KUKA KRL program: MyProgram_003().src

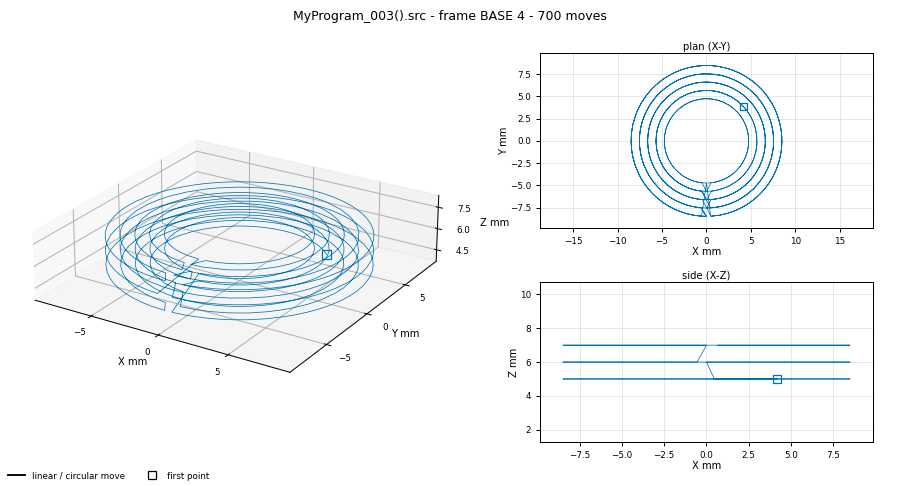
[picture p0: tool path of MyProgram_003().src in frame BASE 4, 700 of 700 moves have a stored position in this frame; points joined in program order, loops and branches not executed]
&ACCESS RVP
&REL 1
&PARAM TEMPLATE = C:\KRC\Roboter\Template\vorgabe
&PARAM EDITMASK = *
DEF MyProgram_003()
; ---- Setting reference (Base) ----
$BASE = BASE_DATA[4]

; --------------------------
; ---- Setting tool (TCP) ----
$TOOL = TOOL_DATA[3]
; --------------------------

$VEL.CP = VEL_APROX_PRINT
Startdeposition()
$VEL.CP = VEL_PRINT
LIN {X 4.1608,Y 3.8743,Z 5,A -2.5016,B 0,C 0,E1 0.1598,E2 90.072} C_DIS
LIN {X 3.5816,Y 4.4156,Z 5,A -2.5001,B 0,C 0,E1 0.1598,E2 90.072} C_DIS
LIN {X 2.9315,Y 4.8693,Z 5,A -2.5049,B 0,C 0,E1 0.1598,E2 90.0721} C_DIS
LIN {X 2.2263,Y 5.2312,Z 5,A -2.5157,B 0,C 0,E1 0.1598,E2 90.0721} C_DIS
LIN {X 1.4771,Y 5.4901,Z 5,A -2.5324,B 0,C 0,E1 0.1598,E2 90.0721} C_DIS
LIN {X 0.6988,Y 5.6397,Z 5,A -2.5548,B 0,C 0,E1 0.1598,E2 90.0721} C_DIS
LIN {X -0.0924,Y 5.6815,Z 5,A -2.5823,B 0,C 0,E1 0.1598,E2 90.0721} C_DIS
LIN {X -0.8823,Y 5.6159,Z 5,A -2.6142,B 0,C 0,E1 0.1598,E2 90.0721} C_DIS
LIN {X -1.6551,Y 5.4395,Z 5,A -2.6501,B 0,C 0,E1 0.1598,E2 90.0721} C_DIS
LIN {X -2.3959,Y 5.1568,Z 5,A -2.6893,B 0,C 0,E1 0.1598,E2 90.072} C_DIS
LIN {X -3.0893,Y 4.7724,Z 5,A -2.7311,B 0,C 0,E1 0.1598,E2 90.0719} C_DIS
LIN {X -3.8738,Y 4.1671,Z 5,A -2.7853,B 0,C 0,E1 0.1598,E2 90.0717} C_DIS
LIN {X -4.6268,Y 3.3119,Z 5,A -2.8489,B 0,C 0,E1 0.1598,E2 90.0714} C_DIS
LIN {X -5.1518,Y 2.4055,Z 5,A -2.9064,B 0,C 0,E1 0.1598,E2 90.0714} C_DIS
LIN {X -5.5303,Y 1.34,Z 5,A -2.965,B 0,C 0,E1 0.1598,E2 90.0711} C_DIS
LIN {X -5.6376,Y 0.726,Z 5,A -2.9951,B 0,C 0,E1 0.1598,E2 90.0713} C_DIS
LIN {X -5.6838,Y -0.1031,Z 5,A -3.0316,B 0,C 0,E1 0.1598,E2 90.0712} C_DIS
LIN {X -5.609,Y -0.9301,Z 5,A -3.0637,B 0,C 0,E1 0.1598,E2 90.0712} C_DIS
LIN {X -5.4131,Y -1.7371,Z 5,A -3.0905,B 0,C 0,E1 0.1598,E2 90.0712} C_DIS
LIN {X -5.1008,Y -2.5065,Z 5,A -3.1115,B 0,C 0,E1 0.1598,E2 90.0712} C_DIS
LIN {X -4.6803,Y -3.2223,Z 5,A -3.1262,B 0,C 0,E1 0.1598,E2 90.0712} C_DIS
LIN {X -4.1611,Y -3.8701,Z 5,A -3.1345,B 0,C 0,E1 0.1598,E2 90.0712} C_DIS
LIN {X -3.3929,Y -4.5678,Z 5,A -3.1357,B 0,C 0,E1 0.1598,E2 90.0711} C_DIS
LIN {X -2.2029,Y -5.2456,Z 5,A -3.1207,B 0,C 0,E1 0.1598,E2 90.0711} C_DIS
LIN {X -1.3096,Y -5.5324,Z 5,A -3.1002,B 0,C 0,E1 0.1598,E2 90.0714} C_DIS
LIN {X -0.5693,Y -5.6561,Z 5,A -3.0783,B 0,C 0,E1 0.1598,E2 90.0714} C_DIS
LIN {X -0.5693,Y -5.6561,Z 5,A -3.0783,B 0,C 0,E1 0.1598,E2 90.0714} C_DIS
Enddeposition()
LIN {X -0.0404,Y -6.6236,Z 5,A -3.0988,B 0,C 0,E1 0.1598,E2 90.0703} C_DIS
Startdeposition()
$VEL.CP = VEL_PRINT
LIN {X -0.9259,Y -6.553,Z 5,A -3.1294,B 0,C 0,E1 0.1598,E2 90.0713} C_DIS
LIN {X -1.6231,Y -6.4161,Z 5,A -3.1492,B 0,C 0,E1 0.1598,E2 90.0713} C_DIS
LIN {X -2.3026,Y -6.2076,Z 5,A -3.1654,B 0,C 0,E1 0.1598,E2 90.0713} C_DIS
LIN {X -2.9544,Y -5.9244,Z 5,A -3.1773,B 0,C 0,E1 0.1598,E2 90.0713} C_DIS
LIN {X -3.5722,Y -5.5732,Z 5,A -3.1851,B 0,C 0,E1 0.1598,E2 90.0713} C_DIS
LIN {X -4.1491,Y -5.1583,Z 5,A -3.1887,B 0,C 0,E1 0.1598,E2 90.0713} C_DIS
LIN {X -4.6779,Y -4.6835,Z 5,A -3.1881,B 0,C 0,E1 0.1598,E2 90.0713} C_DIS
LIN {X -5.1529,Y -4.1549,Z 5,A -3.1832,B 0,C 0,E1 0.1598,E2 90.0712} C_DIS
LIN {X -5.5689,Y -3.5788,Z 5,A -3.1742,B 0,C 0,E1 0.1598,E2 90.0712} C_DIS
LIN {X -5.9215,Y -2.9616,Z 5,A -3.1611,B 0,C 0,E1 0.1598,E2 90.0712} C_DIS
LIN {X -6.202,Y -2.3087,Z 5,A -3.1439,B 0,C 0,E1 0.1598,E2 90.0712} C_DIS
LIN {X -6.4151,Y -1.6307,Z 5,A -3.1231,B 0,C 0,E1 0.1598,E2 90.0712} C_DIS
LIN {X -6.5528,Y -0.9336,Z 5,A -3.0988,B 0,C 0,E1 0.1598,E2 90.0712} C_DIS
LIN {X -6.6173,Y -0.2258,Z 5,A -3.0714,B 0,C 0,E1 0.1598,E2 90.0712} C_DIS
LIN {X -6.6026,Y 0.4846,Z 5,A -3.041,B 0,C 0,E1 0.1598,E2 90.0712} C_DIS
LIN {X -6.5102,Y 1.1893,Z 5,A -3.0079,B 0,C 0,E1 0.1598,E2 90.0713} C_DIS
LIN {X -6.3462,Y 1.8807,Z 5,A -2.9728,B 0,C 0,E1 0.1598,E2 90.0713} C_DIS
LIN {X -6.1101,Y 2.5511,Z 5,A -2.9359,B 0,C 0,E1 0.1598,E2 90.0714} C_DIS
LIN {X -5.8024,Y 3.1918,Z 5,A -2.8976,B 0,C 0,E1 0.1598,E2 90.0715} C_DIS
LIN {X -5.4264,Y 3.795,Z 5,A -2.8584,B 0,C 0,E1 0.1598,E2 90.0715} C_DIS
LIN {X -4.9862,Y 4.3528,Z 5,A -2.8187,B 0,C 0,E1 0.1598,E2 90.0717} C_DIS
LIN {X -4.4919,Y 4.8634,Z 5,A -2.779,B 0,C 0,E1 0.1598,E2 90.0717} C_DIS
LIN {X -3.9448,Y 5.317,Z 5,A -2.7398,B 0,C 0,E1 0.1598,E2 90.0718} C_DIS
LIN {X -3.3521,Y 5.7091,Z 5,A -2.7015,B 0,C 0,E1 0.1598,E2 90.0718} C_DIS
LIN {X -2.7203,Y 6.034,Z 5,A -2.6645,B 0,C 0,E1 0.1598,E2 90.072} C_DIS
LIN {X -2.0578,Y 6.2916,Z 5,A -2.6292,B 0,C 0,E1 0.1598,E2 90.072} C_DIS
LIN {X -1.372,Y 6.4783,Z 5,A -2.596,B 0,C 0,E1 0.1598,E2 90.072} C_DIS
LIN {X -0.6697,Y 6.587,Z 5,A -2.5656,B 0,C 0,E1 0.1598,E2 90.0721} C_DIS
LIN {X 0.0402,Y 6.6208,Z 5,A -2.5379,B 0,C 0,E1 0.1598,E2 90.0721} C_DIS
LIN {X 0.7496,Y 6.5788,Z 5,A -2.5135,B 0,C 0,E1 0.1598,E2 90.0722} C_DIS
LIN {X 1.4503,Y 6.4593,Z 5,A -2.4927,B 0,C 0,E1 0.1598,E2 90.0722} C_DIS
LIN {X 2.1342,Y 6.2657,Z 5,A -2.4756,B 0,C 0,E1 0.1598,E2 90.0722} C_DIS
LIN {X 2.7941,Y 6.0022,Z 5,A -2.4624,B 0,C 0,E1 0.1598,E2 90.0722} C_DIS
LIN {X 3.4211,Y 5.6677,Z 5,A -2.4534,B 0,C 0,E1 0.1598,E2 90.0722} C_DIS
LIN {X 4.0075,Y 5.2662,Z 5,A -2.4487,B 0,C 0,E1 0.1598,E2 90.0722} C_DIS
LIN {X 4.5492,Y 4.8063,Z 5,A -2.4481,B 0,C 0,E1 0.1598,E2 90.0722} C_DIS
LIN {X 5.0416,Y 4.2938,Z 5,A -2.4516,B 0,C 0,E1 0.1598,E2 90.0722} C_DIS
LIN {X 5.4696,Y 3.7264,Z 5,A -2.4598,B 0,C 0,E1 0.1598,E2 90.0722} C_DIS
LIN {X 5.8381,Y 3.1188,Z 5,A -2.4719,B 0,C 0,E1 0.1598,E2 90.0721} C_DIS
LIN {X 6.1397,Y 2.4754,Z 5,A -2.4881,B 0,C 0,E1 0.1598,E2 90.0721} C_DIS
LIN {X 6.3699,Y 1.8031,Z 5,A -2.508,B 0,C 0,E1 0.1598,E2 90.072} C_DIS
LIN {X 6.5278,Y 1.1101,Z 5,A -2.5316,B 0,C 0,E1 0.1598,E2 90.072} C_DIS
LIN {X 6.6079,Y 0.4039,Z 5,A -2.5586,B 0,C 0,E1 0.1598,E2 90.0719} C_DIS
LIN {X 6.6124,Y -0.3068,Z 5,A -2.5885,B 0,C 0,E1 0.1598,E2 90.0719} C_DIS
LIN {X 6.542,Y -1.0138,Z 5,A -2.6211,B 0,C 0,E1 0.1598,E2 90.0719} C_DIS
LIN {X 6.3948,Y -1.7092,Z 5,A -2.656,B 0,C 0,E1 0.1598,E2 90.0718} C_DIS
LIN {X 6.1754,Y -2.3851,Z 5,A -2.6928,B 0,C 0,E1 0.1598,E2 90.0718} C_DIS
LIN {X 5.884,Y -3.0334,Z 5,A -2.731,B 0,C 0,E1 0.1598,E2 90.0718} C_DIS
LIN {X 5.5246,Y -3.6466,Z 5,A -2.7702,B 0,C 0,E1 0.1598,E2 90.0717} C_DIS
LIN {X 5.1021,Y -4.2181,Z 5,A -2.81,B 0,C 0,E1 0.1598,E2 90.0717} C_DIS
LIN {X 4.6202,Y -4.7402,Z 5,A -2.8499,B 0,C 0,E1 0.1598,E2 90.0717} C_DIS
LIN {X 4.0856,Y -5.2087,Z 5,A -2.8894,B 0,C 0,E1 0.1598,E2 90.0717} C_DIS
LIN {X 3.5047,Y -5.6183,Z 5,A -2.9281,B 0,C 0,E1 0.1598,E2 90.0716} C_DIS
LIN {X 2.8824,Y -5.9615,Z 5,A -2.9655,B 0,C 0,E1 0.1598,E2 90.0716} C_DIS
LIN {X 2.2263,Y -6.2348,Z 5,A -3.0012,B 0,C 0,E1 0.1598,E2 90.0716} C_DIS
LIN {X 1.5451,Y -6.4376,Z 5,A -3.0348,B 0,C 0,E1 0.1598,E2 90.0716} C_DIS
LIN {X 0.846,Y -6.5644,Z 5,A -3.0658,B 0,C 0,E1 0.1598,E2 90.0715} C_DIS
LIN {X -0.0404,Y -6.6236,Z 5,A -3.1008,B 0,C 0,E1 0.1598,E2 90.0715} C_DIS
Enddeposition()
LIN {X -0.0404,Y -6.6236,Z 5,A -3.1008,B 0,C 0,E1 0.1598,E2 90.0715} C_DIS
Startdeposition()
$VEL.CP = VEL_PRINT
LIN {X 0.4586,Y -7.5414,Z 5,A -3.121,B 0,C 0,E1 0.1598,E2 90.0709} C_DIS
LIN {X 1.4877,Y -7.4091,Z 5,A -3.0782,B 0,C 0,E1 0.1598,E2 90.0714} C_DIS
LIN {X 2.3467,Y -7.1836,Z 5,A -3.0371,B 0,C 0,E1 0.1598,E2 90.0715} C_DIS
LIN {X 3.457,Y -6.7151,Z 5,A -2.9765,B 0,C 0,E1 0.1598,E2 90.0715} C_DIS
LIN {X 4.4391,Y -6.1176,Z 5,A -2.915,B 0,C 0,E1 0.1598,E2 90.0715} C_DIS
LIN {X 5.3005,Y -5.3806,Z 5,A -2.852,B 0,C 0,E1 0.1598,E2 90.0715} C_DIS
LIN {X 5.8569,Y -4.7686,Z 5,A -2.8057,B 0,C 0,E1 0.1598,E2 90.0716} C_DIS
LIN {X 6.3438,Y -4.0999,Z 5,A -2.7594,B 0,C 0,E1 0.1598,E2 90.0716} C_DIS
LIN {X 6.8478,Y -3.1971,Z 5,A -2.7023,B 0,C 0,E1 0.1598,E2 90.0715} C_DIS
LIN {X 7.2249,Y -2.2147,Z 5,A -2.6467,B 0,C 0,E1 0.1598,E2 90.0715} C_DIS
LIN {X 7.5046,Y -0.888,Z 5,A -2.5797,B 0,C 0,E1 0.1598,E2 90.0712} C_DIS
LIN {X 7.5564,Y 0.1077,Z 5,A -2.536,B 0,C 0,E1 0.1598,E2 90.0717} C_DIS
LIN {X 7.4656,Y 1.1496,Z 5,A -2.495,B 0,C 0,E1 0.1598,E2 90.0717} C_DIS
LIN {X 7.2089,Y 2.2659,Z 5,A -2.4571,B 0,C 0,E1 0.1598,E2 90.0716} C_DIS
LIN {X 6.8696,Y 3.1485,Z 5,A -2.4324,B 0,C 0,E1 0.1598,E2 90.0719} C_DIS
LIN {X 6.2798,Y 4.2042,Z 5,A -2.4093,B 0,C 0,E1 0.1598,E2 90.0718} C_DIS
LIN {X 5.6133,Y 5.0619,Z 5,A -2.3977,B 0,C 0,E1 0.1598,E2 90.0719} C_DIS
LIN {X 4.7836,Y 5.8452,Z 5,A -2.3952,B 0,C 0,E1 0.1598,E2 90.0719} C_DIS
LIN {X 3.9189,Y 6.4611,Z 5,A -2.4012,B 0,C 0,E1 0.1598,E2 90.0721} C_DIS
LIN {X 2.5264,Y 7.1223,Z 5,A -2.4246,B 0,C 0,E1 0.1598,E2 90.0721} C_DIS
LIN {X 1.6107,Y 7.3833,Z 5,A -2.4476,B 0,C 0,E1 0.1598,E2 90.0723} C_DIS
LIN {X -0.1184,Y 7.5562,Z 5,A -2.5042,B 0,C 0,E1 0.1598,E2 90.0723} C_DIS
LIN {X -1.2622,Y 7.4509,Z 5,A -2.5509,B 0,C 0,E1 0.1598,E2 90.0722} C_DIS
LIN {X -2.8172,Y 7.0134,Z 5,A -2.6267,B 0,C 0,E1 0.1598,E2 90.072} C_DIS
LIN {X -3.9999,Y 6.411,Z 5,A -2.6956,B 0,C 0,E1 0.1598,E2 90.0718} C_DIS
LIN {X -4.7613,Y 5.8698,Z 5,A -2.7464,B 0,C 0,E1 0.1598,E2 90.0718} C_DIS
LIN {X -5.6287,Y 5.0444,Z 5,A -2.813,B 0,C 0,E1 0.1598,E2 90.0715} C_DIS
LIN {X -6.3509,Y 4.0973,Z 5,A -2.8793,B 0,C 0,E1 0.1598,E2 90.0713} C_DIS
LIN {X -6.9039,Y 3.0748,Z 5,A -2.9426,B 0,C 0,E1 0.1598,E2 90.0711} C_DIS
LIN {X -7.2823,Y 2.0215,Z 5,A -3.0008,B 0,C 0,E1 0.1598,E2 90.0711} C_DIS
LIN {X -7.4591,Y 1.1875,Z 5,A -3.0426,B 0,C 0,E1 0.1598,E2 90.0711} C_DIS
LIN {X -7.5506,Y 0.3399,Z 5,A -3.0815,B 0,C 0,E1 0.1598,E2 90.0711} C_DIS
LIN {X -7.5339,Y -0.5955,Z 5,A -3.1202,B 0,C 0,E1 0.1598,E2 90.071} C_DIS
LIN {X -7.3478,Y -1.7493,Z 5,A -3.1617,B 0,C 0,E1 0.1598,E2 90.0707} C_DIS
LIN {X -7.0494,Y -2.7246,Z 5,A -3.1919,B 0,C 0,E1 0.1598,E2 90.0707} C_DIS
LIN {X -6.5677,Y -3.731,Z 5,A -3.2166,B 0,C 0,E1 0.1598,E2 90.0707} C_DIS
LIN {X -5.9244,Y -4.6917,Z 5,A -3.2335,B 0,C 0,E1 0.1598,E2 90.0708} C_DIS
LIN {X -5.1075,Y -5.5639,Z 5,A -3.2403,B 0,C 0,E1 0.1598,E2 90.0708} C_DIS
LIN {X -4.2014,Y -6.2818,Z 5,A -3.2375,B 0,C 0,E1 0.1598,E2 90.071} C_DIS
LIN {X -3.3847,Y -6.7567,Z 5,A -3.2278,B 0,C 0,E1 0.1598,E2 90.0712} C_DIS
LIN {X -2.4228,Y -7.1598,Z 5,A -3.2096,B 0,C 0,E1 0.1598,E2 90.0712} C_DIS
LIN {X -1.5721,Y -7.3914,Z 5,A -3.1882,B 0,C 0,E1 0.1598,E2 90.0712} C_DIS
LIN {X -0.6387,Y -7.531,Z 5,A -3.1599,B 0,C 0,E1 0.1598,E2 90.0713} C_DIS
LIN {X -0.6387,Y -7.531,Z 5,A -3.1599,B 0,C 0,E1 0.1598,E2 90.0713} C_DIS
Enddeposition()
LIN {X -0.0485,Y -8.4894,Z 5,A -3.1779,B 0,C 0,E1 0.1598,E2 90.0702} C_DIS
Startdeposition()
$VEL.CP = VEL_PRINT
LIN {X -1.0658,Y -8.4207,Z 5,A -3.2134,B 0,C 0,E1 0.1598,E2 90.0712} C_DIS
LIN {X -1.8694,Y -8.2794,Z 5,A -3.2369,B 0,C 0,E1 0.1598,E2 90.0712} C_DIS
LIN {X -2.6556,Y -8.0613,Z 5,A -3.2565,B 0,C 0,E1 0.1598,E2 90.0712} C_DIS
LIN {X -3.4177,Y -7.7697,Z 5,A -3.2721,B 0,C 0,E1 0.1598,E2 90.0712} C_DIS
LIN {X -4.1482,Y -7.4061,Z 5,A -3.2835,B 0,C 0,E1 0.1598,E2 90.0712} C_DIS
LIN {X -4.8402,Y -6.9737,Z 5,A -3.2906,B 0,C 0,E1 0.1598,E2 90.0711} C_DIS
LIN {X -5.4872,Y -6.4765,Z 5,A -3.2933,B 0,C 0,E1 0.1598,E2 90.0711} C_DIS
LIN {X -6.2257,Y -5.7733,Z 5,A -3.2906,B 0,C 0,E1 0.1598,E2 90.0709} C_DIS
LIN {X -6.9713,Y -4.8425,Z 5,A -3.2785,B 0,C 0,E1 0.1598,E2 90.0707} C_DIS
LIN {X -7.3978,Y -4.1602,Z 5,A -3.2657,B 0,C 0,E1 0.1598,E2 90.071} C_DIS
LIN {X -7.7587,Y -3.441,Z 5,A -3.2486,B 0,C 0,E1 0.1598,E2 90.071} C_DIS
LIN {X -8.0498,Y -2.691,Z 5,A -3.2277,B 0,C 0,E1 0.1598,E2 90.071} C_DIS
LIN {X -8.268,Y -1.9165,Z 5,A -3.2031,B 0,C 0,E1 0.1598,E2 90.071} C_DIS
LIN {X -8.4122,Y -1.125,Z 5,A -3.1751,B 0,C 0,E1 0.1598,E2 90.071} C_DIS
LIN {X -8.4813,Y -0.3234,Z 5,A -3.144,B 0,C 0,E1 0.1598,E2 90.071} C_DIS
LIN {X -8.4491,Y 0.8445,Z 5,A -3.0933,B 0,C 0,E1 0.1598,E2 90.0708} C_DIS
LIN {X -8.2788,Y 1.8895,Z 5,A -3.0432,B 0,C 0,E1 0.1598,E2 90.071} C_DIS
LIN {X -7.9502,Y 2.9764,Z 5,A -2.9854,B 0,C 0,E1 0.1598,E2 90.071} C_DIS
LIN {X -7.621,Y 3.7394,Z 5,A -2.9415,B 0,C 0,E1 0.1598,E2 90.0713} C_DIS
LIN {X -7.2187,Y 4.4667,Z 5,A -2.8961,B 0,C 0,E1 0.1598,E2 90.0714} C_DIS
LIN {X -6.7474,Y 5.151,Z 5,A -2.85,B 0,C 0,E1 0.1598,E2 90.0715} C_DIS
LIN {X -6.2111,Y 5.7858,Z 5,A -2.8036,B 0,C 0,E1 0.1598,E2 90.0716} C_DIS
LIN {X -5.615,Y 6.3648,Z 5,A -2.7573,B 0,C 0,E1 0.1598,E2 90.0717} C_DIS
LIN {X -4.9653,Y 6.8829,Z 5,A -2.7116,B 0,C 0,E1 0.1598,E2 90.0718} C_DIS
LIN {X -4.2682,Y 7.3351,Z 5,A -2.6668,B 0,C 0,E1 0.1598,E2 90.0719} C_DIS
LIN {X -3.5302,Y 7.7169,Z 5,A -2.6235,B 0,C 0,E1 0.1598,E2 90.072} C_DIS
LIN {X -2.7586,Y 8.0253,Z 5,A -2.5821,B 0,C 0,E1 0.1598,E2 90.072} C_DIS
LIN {X -1.9606,Y 8.2567,Z 5,A -2.5429,B 0,C 0,E1 0.1598,E2 90.0722} C_DIS
LIN {X -1.1438,Y 8.4093,Z 5,A -2.5063,B 0,C 0,E1 0.1598,E2 90.0722} C_DIS
LIN {X -0.3161,Y 8.4816,Z 5,A -2.4727,B 0,C 0,E1 0.1598,E2 90.0722} C_DIS
LIN {X 0.5148,Y 8.4729,Z 5,A -2.4424,B 0,C 0,E1 0.1598,E2 90.0723} C_DIS
LIN {X 1.3407,Y 8.3814,Z 5,A -2.4157,B 0,C 0,E1 0.1598,E2 90.0723} C_DIS
LIN {X 2.1537,Y 8.2095,Z 5,A -2.3929,B 0,C 0,E1 0.1598,E2 90.0723} C_DIS
LIN {X 2.9463,Y 7.9598,Z 5,A -2.3742,B 0,C 0,E1 0.1598,E2 90.0723} C_DIS
LIN {X 3.7106,Y 7.6339,Z 5,A -2.3597,B 0,C 0,E1 0.1598,E2 90.0723} C_DIS
LIN {X 4.4394,Y 7.2347,Z 5,A -2.3496,B 0,C 0,E1 0.1598,E2 90.0723} C_DIS
LIN {X 5.3674,Y 6.5808,Z 5,A -2.3429,B 0,C 0,E1 0.1598,E2 90.0722} C_DIS
LIN {X 6.1123,Y 5.8907,Z 5,A -2.3446,B 0,C 0,E1 0.1598,E2 90.0722} C_DIS
LIN {X 6.6465,Y 5.2788,Z 5,A -2.3508,B 0,C 0,E1 0.1598,E2 90.0722} C_DIS
LIN {X 7.1199,Y 4.6188,Z 5,A -2.3613,B 0,C 0,E1 0.1598,E2 90.0722} C_DIS
LIN {X 7.5283,Y 3.9167,Z 5,A -2.376,B 0,C 0,E1 0.1598,E2 90.0722} C_DIS
LIN {X 7.868,Y 3.1789,Z 5,A -2.3947,B 0,C 0,E1 0.1598,E2 90.0721} C_DIS
LIN {X 8.1958,Y 2.2181,Z 5,A -2.4231,B 0,C 0,E1 0.1598,E2 90.0717} C_DIS
LIN {X 8.4199,Y 1.0739,Z 5,A -2.4632,B 0,C 0,E1 0.1598,E2 90.0715} C_DIS
LIN {X 8.4832,Y 0.2891,Z 5,A -2.4946,B 0,C 0,E1 0.1598,E2 90.0719} C_DIS
LIN {X 8.4734,Y -0.4982,Z 5,A -2.5284,B 0,C 0,E1 0.1598,E2 90.0719} C_DIS
LIN {X 8.3355,Y -1.6188,Z 5,A -2.5807,B 0,C 0,E1 0.1598,E2 90.0715} C_DIS
LIN {X 8.077,Y -2.6093,Z 5,A -2.6324,B 0,C 0,E1 0.1598,E2 90.0715} C_DIS
LIN {X 7.7877,Y -3.3754,Z 5,A -2.6757,B 0,C 0,E1 0.1598,E2 90.0717} C_DIS
LIN {X 7.4261,Y -4.1102,Z 5,A -2.7202,B 0,C 0,E1 0.1598,E2 90.0717} C_DIS
LIN {X 6.9956,Y -4.8068,Z 5,A -2.7657,B 0,C 0,E1 0.1598,E2 90.0717} C_DIS
LIN {X 6.5,Y -5.4586,Z 5,A -2.8116,B 0,C 0,E1 0.1598,E2 90.0717} C_DIS
LIN {X 5.7223,Y -6.2741,Z 5,A -2.8746,B 0,C 0,E1 0.1598,E2 90.0714} C_DIS
LIN {X 4.878,Y -6.9455,Z 5,A -2.9342,B 0,C 0,E1 0.1598,E2 90.0714} C_DIS
LIN {X 4.1473,Y -7.4046,Z 5,A -2.9806,B 0,C 0,E1 0.1598,E2 90.0715} C_DIS
LIN {X 3.3736,Y -7.7869,Z 5,A -3.0252,B 0,C 0,E1 0.1598,E2 90.0715} C_DIS
LIN {X 2.5655,Y -8.0896,Z 5,A -3.0677,B 0,C 0,E1 0.1598,E2 90.0715} C_DIS
LIN {X 1.52,Y -8.3549,Z 5,A -3.1172,B 0,C 0,E1 0.1598,E2 90.0714} C_DIS
LIN {X 0.4661,Y -8.4736,Z 5,A -3.1609,B 0,C 0,E1 0.1598,E2 90.0714} C_DIS
LIN {X 0.4661,Y -8.4736,Z 5,A -3.1609,B 0,C 0,E1 0.1598,E2 90.0714} C_DIS
Enddeposition()
LIN {X 0.0002,Y -4.7527,Z 6,A -3.0051,B 0,C 0,E1 0.1598,E2 90.0603} C_DIS
Startdeposition()
$VEL.CP = VEL_PRINT
LIN {X 0.0002,Y -4.7527,Z 6,A -3.0108,B 0,C 0,E1 0.1598,E2 90.066} C_DIS
LIN {X 0.8436,Y -4.6754,Z 6,A -2.9814,B 0,C 0,E1 0.1598,E2 90.0709} C_DIS
LIN {X 1.5802,Y -4.479,Z 6,A -2.9466,B 0,C 0,E1 0.1598,E2 90.0716} C_DIS
LIN {X 2.1262,Y -4.2473,Z 6,A -2.9168,B 0,C 0,E1 0.1598,E2 90.0716} C_DIS
LIN {X 2.7108,Y -3.904,Z 6,A -2.8807,B 0,C 0,E1 0.1598,E2 90.0716} C_DIS
LIN {X 3.2384,Y -3.4779,Z 6,A -2.8433,B 0,C 0,E1 0.1598,E2 90.0716} C_DIS
LIN {X 3.7,Y -2.9815,Z 6,A -2.8052,B 0,C 0,E1 0.1598,E2 90.0717} C_DIS
LIN {X 4.0865,Y -2.4244,Z 6,A -2.7674,B 0,C 0,E1 0.1598,E2 90.0717} C_DIS
LIN {X 4.3892,Y -1.818,Z 6,A -2.7305,B 0,C 0,E1 0.1598,E2 90.0717} C_DIS
LIN {X 4.603,Y -1.1746,Z 6,A -2.6954,B 0,C 0,E1 0.1598,E2 90.0717} C_DIS
LIN {X 4.7242,Y -0.5078,Z 6,A -2.6627,B 0,C 0,E1 0.1598,E2 90.0717} C_DIS
LIN {X 4.7491,Y 0.1698,Z 6,A -2.633,B 0,C 0,E1 0.1598,E2 90.0718} C_DIS
LIN {X 4.6586,Y 0.9268,Z 6,A -2.6042,B 0,C 0,E1 0.1598,E2 90.0718} C_DIS
LIN {X 4.5069,Y 1.5002,Z 6,A -2.5856,B 0,C 0,E1 0.1598,E2 90.0719} C_DIS
LIN {X 4.2491,Y 2.1272,Z 6,A -2.5686,B 0,C 0,E1 0.1598,E2 90.0719} C_DIS
LIN {X 3.9029,Y 2.7102,Z 6,A -2.5567,B 0,C 0,E1 0.1598,E2 90.0719} C_DIS
LIN {X 3.4777,Y 3.2383,Z 6,A -2.55,B 0,C 0,E1 0.1598,E2 90.072} C_DIS
LIN {X 2.9815,Y 3.7002,Z 6,A -2.5488,B 0,C 0,E1 0.1598,E2 90.072} C_DIS
LIN {X 2.4242,Y 4.0861,Z 6,A -2.5531,B 0,C 0,E1 0.1598,E2 90.072} C_DIS
LIN {X 1.8178,Y 4.3889,Z 6,A -2.5627,B 0,C 0,E1 0.1598,E2 90.072} C_DIS
LIN {X 1.1746,Y 4.6027,Z 6,A -2.5774,B 0,C 0,E1 0.1598,E2 90.0721} C_DIS
LIN {X 0.5077,Y 4.7248,Z 6,A -2.5968,B 0,C 0,E1 0.1598,E2 90.0721} C_DIS
LIN {X -0.2544,Y 4.7428,Z 6,A -2.6242,B 0,C 0,E1 0.1598,E2 90.0721} C_DIS
LIN {X -0.8439,Y 4.6769,Z 6,A -2.6487,B 0,C 0,E1 0.1598,E2 90.0721} C_DIS
LIN {X -1.5001,Y 4.5068,Z 6,A -2.6801,B 0,C 0,E1 0.1598,E2 90.072} C_DIS
LIN {X -2.1271,Y 4.249,Z 6,A -2.714,B 0,C 0,E1 0.1598,E2 90.072} C_DIS
LIN {X -2.7104,Y 3.9033,Z 6,A -2.7501,B 0,C 0,E1 0.1598,E2 90.0719} C_DIS
LIN {X -3.2385,Y 3.4781,Z 6,A -2.7874,B 0,C 0,E1 0.1598,E2 90.0718} C_DIS
LIN {X -3.6997,Y 2.9813,Z 6,A -2.8253,B 0,C 0,E1 0.1598,E2 90.0717} C_DIS
LIN {X -4.0859,Y 2.4241,Z 6,A -2.863,B 0,C 0,E1 0.1598,E2 90.0717} C_DIS
LIN {X -4.3885,Y 1.8175,Z 6,A -2.8996,B 0,C 0,E1 0.1598,E2 90.0715} C_DIS
LIN {X -4.6022,Y 1.1744,Z 6,A -2.9346,B 0,C 0,E1 0.1598,E2 90.0715} C_DIS
LIN {X -4.7237,Y 0.5076,Z 6,A -2.9671,B 0,C 0,E1 0.1598,E2 90.0714} C_DIS
LIN {X -4.749,Y -0.1698,Z 6,A -2.9966,B 0,C 0,E1 0.1598,E2 90.0714} C_DIS
LIN {X -4.6753,Y -0.8437,Z 6,A -3.0223,B 0,C 0,E1 0.1598,E2 90.0714} C_DIS
LIN {X -4.5073,Y -1.5004,Z 6,A -3.0438,B 0,C 0,E1 0.1598,E2 90.0713} C_DIS
LIN {X -4.2474,Y -2.1265,Z 6,A -3.0606,B 0,C 0,E1 0.1598,E2 90.0713} C_DIS
LIN {X -3.9034,Y -2.7105,Z 6,A -3.0727,B 0,C 0,E1 0.1598,E2 90.0713} C_DIS
LIN {X -3.4778,Y -3.2384,Z 6,A -3.0793,B 0,C 0,E1 0.1598,E2 90.0713} C_DIS
LIN {X -2.9815,Y -3.7,Z 6,A -3.0806,B 0,C 0,E1 0.1598,E2 90.0713} C_DIS
LIN {X -2.4244,Y -4.0865,Z 6,A -3.0765,B 0,C 0,E1 0.1598,E2 90.0713} C_DIS
LIN {X -1.8178,Y -4.3887,Z 6,A -3.067,B 0,C 0,E1 0.1598,E2 90.0714} C_DIS
LIN {X -1.1745,Y -4.6023,Z 6,A -3.0524,B 0,C 0,E1 0.1598,E2 90.0714} C_DIS
LIN {X -0.5077,Y -4.725,Z 6,A -3.0332,B 0,C 0,E1 0.1598,E2 90.0715} C_DIS
LIN {X -0.5077,Y -4.725,Z 6,A -3.0332,B 0,C 0,E1 0.1598,E2 90.0715} C_DIS
Enddeposition()
LIN {X 0.0016,Y -5.6864,Z 6,A -3.0541,B 0,C 0,E1 0.1598,E2 90.0703} C_DIS
Startdeposition()
$VEL.CP = VEL_PRINT
LIN {X -0.9286,Y -5.6133,Z 6,A -3.0863,B 0,C 0,E1 0.1598,E2 90.0714} C_DIS
LIN {X -2.0374,Y -5.3126,Z 6,A -3.1142,B 0,C 0,E1 0.1598,E2 90.0714} C_DIS
LIN {X -3.1502,Y -4.7386,Z 6,A -3.1307,B 0,C 0,E1 0.1598,E2 90.0712} C_DIS
LIN {X -3.9721,Y -4.0673,Z 6,A -3.1325,B 0,C 0,E1 0.1598,E2 90.0712} C_DIS
LIN {X -4.5331,Y -3.43,Z 6,A -3.1262,B 0,C 0,E1 0.1598,E2 90.0712} C_DIS
LIN {X -4.9939,Y -2.717,Z 6,A -3.1131,B 0,C 0,E1 0.1598,E2 90.0712} C_DIS
LIN {X -5.3425,Y -1.9429,Z 6,A -3.0932,B 0,C 0,E1 0.1598,E2 90.0712} C_DIS
LIN {X -5.5724,Y -1.1256,Z 6,A -3.0672,B 0,C 0,E1 0.1598,E2 90.0712} C_DIS
LIN {X -5.6786,Y -0.2832,Z 6,A -3.0356,B 0,C 0,E1 0.1598,E2 90.0712} C_DIS
LIN {X -5.6579,Y 0.5657,Z 6,A -2.999,B 0,C 0,E1 0.1598,E2 90.0712} C_DIS
LIN {X -5.51,Y 1.4018,Z 6,A -2.9584,B 0,C 0,E1 0.1598,E2 90.0712} C_DIS
LIN {X -5.2388,Y 2.2064,Z 6,A -2.9146,B 0,C 0,E1 0.1598,E2 90.0714} C_DIS
LIN {X -4.852,Y 2.962,Z 6,A -2.8685,B 0,C 0,E1 0.1598,E2 90.0714} C_DIS
LIN {X -4.2219,Y 3.816,Z 6,A -2.8092,B 0,C 0,E1 0.1598,E2 90.0714} C_DIS
LIN {X -3.4205,Y 4.539,Z 6,A -2.7494,B 0,C 0,E1 0.1598,E2 90.0716} C_DIS
LIN {X -2.7779,Y 4.9589,Z 6,A -2.7082,B 0,C 0,E1 0.1598,E2 90.0719} C_DIS
LIN {X -2.0841,Y 5.2875,Z 6,A -2.6688,B 0,C 0,E1 0.1598,E2 90.0719} C_DIS
LIN {X -1.3526,Y 5.52,Z 6,A -2.632,B 0,C 0,E1 0.1598,E2 90.072} C_DIS
LIN {X -0.1317,Y 5.6882,Z 6,A -2.5799,B 0,C 0,E1 0.1598,E2 90.0721} C_DIS
LIN {X 0.8981,Y 5.6176,Z 6,A -2.5449,B 0,C 0,E1 0.1598,E2 90.0721} C_DIS
LIN {X 1.7964,Y 5.3994,Z 6,A -2.5209,B 0,C 0,E1 0.1598,E2 90.0721} C_DIS
LIN {X 2.7265,Y 4.9883,Z 6,A -2.5039,B 0,C 0,E1 0.1598,E2 90.0721} C_DIS
LIN {X 3.4094,Y 4.5466,Z 6,A -2.4974,B 0,C 0,E1 0.1598,E2 90.0721} C_DIS
LIN {X 4.0231,Y 4.0131,Z 6,A -2.4973,B 0,C 0,E1 0.1598,E2 90.0721} C_DIS
LIN {X 4.5559,Y 3.3986,Z 6,A -2.5036,B 0,C 0,E1 0.1598,E2 90.0721} C_DIS
LIN {X 5.0933,Y 2.5357,Z 6,A -2.5201,B 0,C 0,E1 0.1598,E2 90.0717} C_DIS
LIN {X 5.4458,Y 1.6481,Z 6,A -2.5447,B 0,C 0,E1 0.1598,E2 90.0717} C_DIS
LIN {X 5.6762,Y 0.3921,Z 6,A -2.589,B 0,C 0,E1 0.1598,E2 90.0712} C_DIS
LIN {X 5.6646,Y -0.496,Z 6,A -2.6275,B 0,C 0,E1 0.1598,E2 90.0716} C_DIS
LIN {X 5.5334,Y -1.2989,Z 6,A -2.6665,B 0,C 0,E1 0.1598,E2 90.0716} C_DIS
LIN {X 5.2919,Y -2.0756,Z 6,A -2.7083,B 0,C 0,E1 0.1598,E2 90.0716} C_DIS
LIN {X 4.9409,Y -2.8093,Z 6,A -2.7523,B 0,C 0,E1 0.1598,E2 90.0716} C_DIS
LIN {X 4.4886,Y -3.4853,Z 6,A -2.7977,B 0,C 0,E1 0.1598,E2 90.0716} C_DIS
LIN {X 3.9456,Y -4.0907,Z 6,A -2.8433,B 0,C 0,E1 0.1598,E2 90.0716} C_DIS
LIN {X 3.3214,Y -4.6121,Z 6,A -2.8884,B 0,C 0,E1 0.1598,E2 90.0716} C_DIS
LIN {X 2.6283,Y -5.0374,Z 6,A -2.9319,B 0,C 0,E1 0.1598,E2 90.0716} C_DIS
LIN {X 1.5944,Y -5.4618,Z 6,A -2.9878,B 0,C 0,E1 0.1598,E2 90.0716} C_DIS
LIN {X 0.5504,Y -5.6581,Z 6,A -3.0345,B 0,C 0,E1 0.1598,E2 90.0716} C_DIS
LIN {X 0.5504,Y -5.6581,Z 6,A -3.0345,B 0,C 0,E1 0.1598,E2 90.0716} C_DIS
Enddeposition()
LIN {X 0.0383,Y -6.6235,Z 6,A -3.0932,B 0,C 0,E1 0.1598,E2 90.0703} C_DIS
Startdeposition()
$VEL.CP = VEL_PRINT
LIN {X 0.902,Y -6.5573,Z 6,A -3.0598,B 0,C 0,E1 0.1598,E2 90.0714} C_DIS
LIN {X 1.5828,Y -6.4287,Z 6,A -3.0294,B 0,C 0,E1 0.1598,E2 90.0715} C_DIS
LIN {X 2.246,Y -6.2279,Z 6,A -2.9966,B 0,C 0,E1 0.1598,E2 90.0715} C_DIS
LIN {X 2.8852,Y -5.9601,Z 6,A -2.9617,B 0,C 0,E1 0.1598,E2 90.0715} C_DIS
LIN {X 3.4926,Y -5.6265,Z 6,A -2.9253,B 0,C 0,E1 0.1598,E2 90.0716} C_DIS
LIN {X 4.0598,Y -5.2283,Z 6,A -2.8876,B 0,C 0,E1 0.1598,E2 90.0716} C_DIS
LIN {X 4.5845,Y -4.7755,Z 6,A -2.8491,B 0,C 0,E1 0.1598,E2 90.0716} C_DIS
LIN {X 5.0583,Y -4.2699,Z 6,A -2.8102,B 0,C 0,E1 0.1598,E2 90.0716} C_DIS
LIN {X 5.4775,Y -3.7182,Z 6,A -2.7714,B 0,C 0,E1 0.1598,E2 90.0717} C_DIS
LIN {X 5.8343,Y -3.1241,Z 6,A -2.733,B 0,C 0,E1 0.1598,E2 90.0717} C_DIS
LIN {X 6.1302,Y -2.4976,Z 6,A -2.6956,B 0,C 0,E1 0.1598,E2 90.0717} C_DIS
LIN {X 6.358,Y -1.8433,Z 6,A -2.6594,B 0,C 0,E1 0.1598,E2 90.0717} C_DIS
LIN {X 6.5159,Y -1.1686,Z 6,A -2.625,B 0,C 0,E1 0.1598,E2 90.0718} C_DIS
LIN {X 6.6029,Y -0.481,Z 6,A -2.5926,B 0,C 0,E1 0.1598,E2 90.0718} C_DIS
LIN {X 6.6153,Y 0.2117,Z 6,A -2.5627,B 0,C 0,E1 0.1598,E2 90.0718} C_DIS
LIN {X 6.5589,Y 0.9023,Z 6,A -2.5355,B 0,C 0,E1 0.1598,E2 90.0719} C_DIS
LIN {X 6.4286,Y 1.5828,Z 6,A -2.5115,B 0,C 0,E1 0.1598,E2 90.0719} C_DIS
LIN {X 6.2279,Y 2.2461,Z 6,A -2.4908,B 0,C 0,E1 0.1598,E2 90.072} C_DIS
LIN {X 5.9594,Y 2.8849,Z 6,A -2.4736,B 0,C 0,E1 0.1598,E2 90.072} C_DIS
LIN {X 5.6235,Y 3.491,Z 6,A -2.4603,B 0,C 0,E1 0.1598,E2 90.072} C_DIS
LIN {X 5.2272,Y 4.0593,Z 6,A -2.4509,B 0,C 0,E1 0.1598,E2 90.0721} C_DIS
LIN {X 4.7768,Y 4.5859,Z 6,A -2.4452,B 0,C 0,E1 0.1598,E2 90.0721} C_DIS
LIN {X 4.2705,Y 5.0592,Z 6,A -2.4439,B 0,C 0,E1 0.1598,E2 90.0721} C_DIS
LIN {X 3.7171,Y 5.4764,Z 6,A -2.4467,B 0,C 0,E1 0.1598,E2 90.0722} C_DIS
LIN {X 3.1238,Y 5.8341,Z 6,A -2.4535,B 0,C 0,E1 0.1598,E2 90.0722} C_DIS
LIN {X 2.498,Y 6.1314,Z 6,A -2.464,B 0,C 0,E1 0.1598,E2 90.0722} C_DIS
LIN {X 1.8434,Y 6.3588,Z 6,A -2.4786,B 0,C 0,E1 0.1598,E2 90.0722} C_DIS
LIN {X 1.1685,Y 6.5152,Z 6,A -2.4969,B 0,C 0,E1 0.1598,E2 90.0722} C_DIS
LIN {X 0.481,Y 6.603,Z 6,A -2.5186,B 0,C 0,E1 0.1598,E2 90.0722} C_DIS
LIN {X -0.2117,Y 6.618,Z 6,A -2.5436,B 0,C 0,E1 0.1598,E2 90.0722} C_DIS
LIN {X -0.9022,Y 6.5592,Z 6,A -2.5715,B 0,C 0,E1 0.1598,E2 90.0722} C_DIS
LIN {X -1.5829,Y 6.4292,Z 6,A -2.6021,B 0,C 0,E1 0.1598,E2 90.0721} C_DIS
LIN {X -2.2454,Y 6.2265,Z 6,A -2.6351,B 0,C 0,E1 0.1598,E2 90.0721} C_DIS
LIN {X -2.884,Y 5.9576,Z 6,A -2.67,B 0,C 0,E1 0.1598,E2 90.072} C_DIS
LIN {X -3.4927,Y 5.6265,Z 6,A -2.7063,B 0,C 0,E1 0.1598,E2 90.072} C_DIS
LIN {X -4.0602,Y 5.2288,Z 6,A -2.744,B 0,C 0,E1 0.1598,E2 90.0718} C_DIS
LIN {X -4.5838,Y 4.7747,Z 6,A -2.7824,B 0,C 0,E1 0.1598,E2 90.0718} C_DIS
LIN {X -5.06,Y 4.2713,Z 6,A -2.8211,B 0,C 0,E1 0.1598,E2 90.0717} C_DIS
LIN {X -5.4785,Y 3.719,Z 6,A -2.8598,B 0,C 0,E1 0.1598,E2 90.0717} C_DIS
LIN {X -5.837,Y 3.1259,Z 6,A -2.8979,B 0,C 0,E1 0.1598,E2 90.0715} C_DIS
LIN {X -6.1312,Y 2.4986,Z 6,A -2.9351,B 0,C 0,E1 0.1598,E2 90.0715} C_DIS
LIN {X -6.3578,Y 1.8438,Z 6,A -2.971,B 0,C 0,E1 0.1598,E2 90.0714} C_DIS
LIN {X -6.5154,Y 1.169,Z 6,A -3.0052,B 0,C 0,E1 0.1598,E2 90.0714} C_DIS
LIN {X -6.6036,Y 0.4816,Z 6,A -3.0373,B 0,C 0,E1 0.1598,E2 90.0713} C_DIS
LIN {X -6.6181,Y -0.2111,Z 6,A -3.067,B 0,C 0,E1 0.1598,E2 90.0713} C_DIS
LIN {X -6.5587,Y -0.9016,Z 6,A -3.0939,B 0,C 0,E1 0.1598,E2 90.0713} C_DIS
LIN {X -6.4284,Y -1.5821,Z 6,A -3.1178,B 0,C 0,E1 0.1598,E2 90.0712} C_DIS
LIN {X -6.2281,Y -2.2455,Z 6,A -3.1383,B 0,C 0,E1 0.1598,E2 90.0712} C_DIS
LIN {X -5.9584,Y -2.8837,Z 6,A -3.1553,B 0,C 0,E1 0.1598,E2 90.0712} C_DIS
LIN {X -5.6232,Y -3.4901,Z 6,A -3.1686,B 0,C 0,E1 0.1598,E2 90.0712} C_DIS
LIN {X -5.2276,Y -4.059,Z 6,A -3.1781,B 0,C 0,E1 0.1598,E2 90.0712} C_DIS
LIN {X -4.7744,Y -4.5831,Z 6,A -3.1836,B 0,C 0,E1 0.1598,E2 90.0712} C_DIS
LIN {X -4.2715,Y -5.0598,Z 6,A -3.1852,B 0,C 0,E1 0.1598,E2 90.0712} C_DIS
LIN {X -3.7187,Y -5.4778,Z 6,A -3.1826,B 0,C 0,E1 0.1598,E2 90.0712} C_DIS
LIN {X -3.1248,Y -5.8349,Z 6,A -3.1759,B 0,C 0,E1 0.1598,E2 90.0712} C_DIS
LIN {X -2.4974,Y -6.129,Z 6,A -3.1653,B 0,C 0,E1 0.1598,E2 90.0713} C_DIS
LIN {X -1.8434,Y -6.3575,Z 6,A -3.151,B 0,C 0,E1 0.1598,E2 90.0713} C_DIS
LIN {X -1.1687,Y -6.515,Z 6,A -3.1329,B 0,C 0,E1 0.1598,E2 90.0713} C_DIS
LIN {X -0.4812,Y -6.6017,Z 6,A -3.1114,B 0,C 0,E1 0.1598,E2 90.0714} C_DIS
LIN {X -0.4812,Y -6.6017,Z 6,A -3.1114,B 0,C 0,E1 0.1598,E2 90.0714} C_DIS
Enddeposition()
LIN {X 0.0321,Y -7.5538,Z 6,A -3.1319,B 0,C 0,E1 0.1598,E2 90.0703} C_DIS
Startdeposition()
$VEL.CP = VEL_PRINT
LIN {X -0.8322,Y -7.5109,Z 6,A -3.1629,B 0,C 0,E1 0.1598,E2 90.0713} C_DIS
LIN {X -2.0906,Y -7.2637,Z 6,A -3.1986,B 0,C 0,E1 0.1598,E2 90.0713} C_DIS
LIN {X -2.9095,Y -6.9742,Z 6,A -3.2163,B 0,C 0,E1 0.1598,E2 90.0713} C_DIS
LIN {X -3.8004,Y -6.5275,Z 6,A -3.2301,B 0,C 0,E1 0.1598,E2 90.0712} C_DIS
LIN {X -4.4675,Y -6.0907,Z 6,A -3.2361,B 0,C 0,E1 0.1598,E2 90.0712} C_DIS
LIN {X -5.0842,Y -5.5853,Z 6,A -3.2374,B 0,C 0,E1 0.1598,E2 90.0712} C_DIS
LIN {X -5.6447,Y -5.0182,Z 6,A -3.234,B 0,C 0,E1 0.1598,E2 90.0711} C_DIS
LIN {X -6.2594,Y -4.2338,Z 6,A -3.2233,B 0,C 0,E1 0.1598,E2 90.0709} C_DIS
LIN {X -6.8023,Y -3.2909,Z 6,A -3.2034,B 0,C 0,E1 0.1598,E2 90.0709} C_DIS
LIN {X -7.1688,Y -2.378,Z 6,A -3.1785,B 0,C 0,E1 0.1598,E2 90.0709} C_DIS
LIN {X -7.4555,Y -1.2334,Z 6,A -3.1406,B 0,C 0,E1 0.1598,E2 90.0707} C_DIS
LIN {X -7.558,Y 0.0366,Z 6,A -3.0908,B 0,C 0,E1 0.1598,E2 90.0707} C_DIS
LIN {X -7.4768,Y 1.0699,Z 6,A -3.0446,B 0,C 0,E1 0.1598,E2 90.071} C_DIS
LIN {X -7.2362,Y 2.1788,Z 6,A -2.989,B 0,C 0,E1 0.1598,E2 90.071} C_DIS
LIN {X -6.9059,Y 3.0701,Z 6,A -2.9395,B 0,C 0,E1 0.1598,E2 90.0712} C_DIS
LIN {X -6.0801,Y 4.4894,Z 6,A -2.8489,B 0,C 0,E1 0.1598,E2 90.0708} C_DIS
LIN {X -5.2325,Y 5.4518,Z 6,A -2.7776,B 0,C 0,E1 0.1598,E2 90.0714} C_DIS
LIN {X -4.4836,Y 6.084,Z 6,A -2.7237,B 0,C 0,E1 0.1598,E2 90.0718} C_DIS
LIN {X -3.2599,Y 6.8173,Z 6,A -2.6476,B 0,C 0,E1 0.1598,E2 90.0718} C_DIS
LIN {X -2.4976,Y 7.1329,Z 6,A -2.6063,B 0,C 0,E1 0.1598,E2 90.072} C_DIS
LIN {X -1.4191,Y 7.4235,Z 6,A -2.5543,B 0,C 0,E1 0.1598,E2 90.0721} C_DIS
LIN {X -0.2543,Y 7.5486,Z 6,A -2.5061,B 0,C 0,E1 0.1598,E2 90.0722} C_DIS
LIN {X 0.8744,Y 7.5061,Z 6,A -2.4662,B 0,C 0,E1 0.1598,E2 90.0722} C_DIS
LIN {X 1.7434,Y 7.3545,Z 6,A -2.4405,B 0,C 0,E1 0.1598,E2 90.0722} C_DIS
LIN {X 2.976,Y 6.9459,Z 6,A -2.4121,B 0,C 0,E1 0.1598,E2 90.0722} C_DIS
LIN {X 4.143,Y 6.3219,Z 6,A -2.3953,B 0,C 0,E1 0.1598,E2 90.0722} C_DIS
LIN {X 5.1524,Y 5.5278,Z 6,A -2.3915,B 0,C 0,E1 0.1598,E2 90.072} C_DIS
LIN {X 5.8888,Y 4.7277,Z 6,A -2.3983,B 0,C 0,E1 0.1598,E2 90.072} C_DIS
LIN {X 6.7057,Y 3.4876,Z 6,A -2.42,B 0,C 0,E1 0.1598,E2 90.0714} C_DIS
LIN {X 7.2534,Y 2.1238,Z 6,A -2.4576,B 0,C 0,E1 0.1598,E2 90.0713} C_DIS
LIN {X 7.483,Y 1.0287,Z 6,A -2.4959,B 0,C 0,E1 0.1598,E2 90.0715} C_DIS
LIN {X 7.5495,Y 0.2728,Z 6,A -2.5259,B 0,C 0,E1 0.1598,E2 90.0719} C_DIS
LIN {X 7.5053,Y -0.8816,Z 6,A -2.5761,B 0,C 0,E1 0.1598,E2 90.0714} C_DIS
LIN {X 7.2958,Y -1.9694,Z 6,A -2.6301,B 0,C 0,E1 0.1598,E2 90.0714} C_DIS
LIN {X 6.9033,Y -3.0657,Z 6,A -2.691,B 0,C 0,E1 0.1598,E2 90.0714} C_DIS
LIN {X 6.5158,Y -3.8192,Z 6,A -2.7375,B 0,C 0,E1 0.1598,E2 90.0716} C_DIS
LIN {X 6.0473,Y -4.5252,Z 6,A -2.7848,B 0,C 0,E1 0.1598,E2 90.0716} C_DIS
LIN {X 5.2946,Y -5.3928,Z 6,A -2.8491,B 0,C 0,E1 0.1598,E2 90.0714} C_DIS
LIN {X 4.444,Y -6.1062,Z 6,A -2.9107,B 0,C 0,E1 0.1598,E2 90.0714} C_DIS
LIN {X 3.5041,Y -6.6967,Z 6,A -2.9703,B 0,C 0,E1 0.1598,E2 90.0714} C_DIS
LIN {X 2.61,Y -7.0915,Z 6,A -3.0199,B 0,C 0,E1 0.1598,E2 90.0714} C_DIS
LIN {X 1.6498,Y -7.3751,Z 6,A -3.0672,B 0,C 0,E1 0.1598,E2 90.0714} C_DIS
LIN {X 0.7225,Y -7.5208,Z 6,A -3.1074,B 0,C 0,E1 0.1598,E2 90.0714} C_DIS
LIN {X 0.0321,Y -7.5538,Z 6,A -3.1341,B 0,C 0,E1 0.1598,E2 90.0714} C_DIS
Enddeposition()
LIN {X 0.0321,Y -7.5538,Z 6,A -3.1341,B 0,C 0,E1 0.1598,E2 90.0714} C_DIS
Startdeposition()
$VEL.CP = VEL_PRINT
LIN {X 0.503,Y -8.4716,Z 6,A -3.1554,B 0,C 0,E1 0.1598,E2 90.0708} C_DIS
LIN {X 1.5211,Y -8.3547,Z 6,A -3.1136,B 0,C 0,E1 0.1598,E2 90.0714} C_DIS
LIN {X 2.4577,Y -8.1271,Z 6,A -3.0696,B 0,C 0,E1 0.1598,E2 90.0714} C_DIS
LIN {X 3.4386,Y -7.76,Z 6,A -3.0181,B 0,C 0,E1 0.1598,E2 90.0714} C_DIS
LIN {X 4.187,Y -7.3834,Z 6,A -2.9746,B 0,C 0,E1 0.1598,E2 90.0715} C_DIS
LIN {X 4.8945,Y -6.9344,Z 6,A -2.9296,B 0,C 0,E1 0.1598,E2 90.0715} C_DIS
LIN {X 5.5548,Y -6.4186,Z 6,A -2.8835,B 0,C 0,E1 0.1598,E2 90.0716} C_DIS
LIN {X 6.161,Y -5.8402,Z 6,A -2.8366,B 0,C 0,E1 0.1598,E2 90.0716} C_DIS
LIN {X 6.7068,Y -5.2044,Z 6,A -2.7896,B 0,C 0,E1 0.1598,E2 90.0716} C_DIS
LIN {X 7.1868,Y -4.5176,Z 6,A -2.7427,B 0,C 0,E1 0.1598,E2 90.0716} C_DIS
LIN {X 7.5968,Y -3.7869,Z 6,A -2.6966,B 0,C 0,E1 0.1598,E2 90.0716} C_DIS
LIN {X 7.9331,Y -3.0194,Z 6,A -2.6516,B 0,C 0,E1 0.1598,E2 90.0717} C_DIS
LIN {X 8.1923,Y -2.2226,Z 6,A -2.6082,B 0,C 0,E1 0.1598,E2 90.0717} C_DIS
LIN {X 8.4226,Y -1.0778,Z 6,A -2.5508,B 0,C 0,E1 0.1598,E2 90.0715} C_DIS
LIN {X 8.4875,Y -0.0986,Z 6,A -2.507,B 0,C 0,E1 0.1598,E2 90.0717} C_DIS
LIN {X 8.4603,Y 0.6859,Z 6,A -2.4748,B 0,C 0,E1 0.1598,E2 90.0719} C_DIS
LIN {X 8.3273,Y 1.6583,Z 6,A -2.4382,B 0,C 0,E1 0.1598,E2 90.0717} C_DIS
LIN {X 8.0203,Y 2.7727,Z 6,A -2.4021,B 0,C 0,E1 0.1598,E2 90.0717} C_DIS
LIN {X 7.7083,Y 3.5488,Z 6,A -2.381,B 0,C 0,E1 0.1598,E2 90.072} C_DIS
LIN {X 7.3216,Y 4.2905,Z 6,A -2.3639,B 0,C 0,E1 0.1598,E2 90.072} C_DIS
LIN {X 6.8639,Y 4.9906,Z 6,A -2.3511,B 0,C 0,E1 0.1598,E2 90.0721} C_DIS
LIN {X 6.3397,Y 5.6423,Z 6,A -2.3429,B 0,C 0,E1 0.1598,E2 90.0721} C_DIS
LIN {X 5.754,Y 6.2395,Z 6,A -2.3393,B 0,C 0,E1 0.1598,E2 90.0722} C_DIS
LIN {X 5.1121,Y 6.7758,Z 6,A -2.3403,B 0,C 0,E1 0.1598,E2 90.0722} C_DIS
LIN {X 4.4197,Y 7.2451,Z 6,A -2.3461,B 0,C 0,E1 0.1598,E2 90.0723} C_DIS
LIN {X 3.6848,Y 7.6444,Z 6,A -2.3563,B 0,C 0,E1 0.1598,E2 90.0723} C_DIS
LIN {X 2.9146,Y 7.9706,Z 6,A -2.371,B 0,C 0,E1 0.1598,E2 90.0723} C_DIS
LIN {X 2.1159,Y 8.219,Z 6,A -2.3901,B 0,C 0,E1 0.1598,E2 90.0723} C_DIS
LIN {X 1.2967,Y 8.3879,Z 6,A -2.4132,B 0,C 0,E1 0.1598,E2 90.0723} C_DIS
LIN {X 0.4649,Y 8.4751,Z 6,A -2.4403,B 0,C 0,E1 0.1598,E2 90.0723} C_DIS
LIN {X -0.3715,Y 8.4786,Z 6,A -2.471,B 0,C 0,E1 0.1598,E2 90.0723} C_DIS
LIN {X -1.2042,Y 8.4001,Z 6,A -2.5051,B 0,C 0,E1 0.1598,E2 90.0723} C_DIS
LIN {X -2.0252,Y 8.2404,Z 6,A -2.5421,B 0,C 0,E1 0.1598,E2 90.0722} C_DIS
LIN {X -2.8265,Y 8.0009,Z 6,A -2.5818,B 0,C 0,E1 0.1598,E2 90.0722} C_DIS
LIN {X -3.6004,Y 7.6837,Z 6,A -2.6237,B 0,C 0,E1 0.1598,E2 90.072} C_DIS
LIN {X -4.3393,Y 7.2919,Z 6,A -2.6674,B 0,C 0,E1 0.1598,E2 90.072} C_DIS
LIN {X -5.0363,Y 6.8296,Z 6,A -2.7126,B 0,C 0,E1 0.1598,E2 90.0719} C_DIS
LIN {X -5.6845,Y 6.3011,Z 6,A -2.7587,B 0,C 0,E1 0.1598,E2 90.0718} C_DIS
LIN {X -6.2777,Y 5.7114,Z 6,A -2.8053,B 0,C 0,E1 0.1598,E2 90.0717} C_DIS
LIN {X -6.8096,Y 5.066,Z 6,A -2.8521,B 0,C 0,E1 0.1598,E2 90.0716} C_DIS
LIN {X -7.2752,Y 4.3712,Z 6,A -2.8984,B 0,C 0,E1 0.1598,E2 90.0715} C_DIS
LIN {X -7.6703,Y 3.634,Z 6,A -2.9439,B 0,C 0,E1 0.1598,E2 90.0714} C_DIS
LIN {X -7.9912,Y 2.8615,Z 6,A -2.9882,B 0,C 0,E1 0.1598,E2 90.0713} C_DIS
LIN {X -8.3034,Y 1.7722,Z 6,A -3.0452,B 0,C 0,E1 0.1598,E2 90.071} C_DIS
LIN {X -8.451,Y 0.7776,Z 6,A -3.0925,B 0,C 0,E1 0.1598,E2 90.071} C_DIS
LIN {X -8.4871,Y -0.0261,Z 6,A -3.1278,B 0,C 0,E1 0.1598,E2 90.071} C_DIS
LIN {X -8.4453,Y -0.8295,Z 6,A -3.16,B 0,C 0,E1 0.1598,E2 90.071} C_DIS
LIN {X -8.3291,Y -1.6256,Z 6,A -3.1892,B 0,C 0,E1 0.1598,E2 90.071} C_DIS
LIN {X -8.0218,Y -2.7854,Z 6,A -3.2264,B 0,C 0,E1 0.1598,E2 90.0706} C_DIS
LIN {X -7.5764,Y -3.824,Z 6,A -3.2538,B 0,C 0,E1 0.1598,E2 90.0706} C_DIS
LIN {X -7.1636,Y -4.553,Z 6,A -3.2697,B 0,C 0,E1 0.1598,E2 90.0709} C_DIS
LIN {X -6.68,Y -5.2371,Z 6,A -3.2808,B 0,C 0,E1 0.1598,E2 90.0709} C_DIS
LIN {X -6.1317,Y -5.8706,Z 6,A -3.2874,B 0,C 0,E1 0.1598,E2 90.0709} C_DIS
LIN {X -5.5235,Y -6.4467,Z 6,A -3.2894,B 0,C 0,E1 0.1598,E2 90.071} C_DIS
LIN {X -4.8611,Y -6.9596,Z 6,A -3.2868,B 0,C 0,E1 0.1598,E2 90.071} C_DIS
LIN {X -4.1512,Y -7.4044,Z 6,A -3.2796,B 0,C 0,E1 0.1598,E2 90.071} C_DIS
LIN {X -3.4009,Y -7.7774,Z 6,A -3.2678,B 0,C 0,E1 0.1598,E2 90.0711} C_DIS
LIN {X -2.273,Y -8.1815,Z 6,A -3.2436,B 0,C 0,E1 0.1598,E2 90.0711} C_DIS
LIN {X -1.3284,Y -8.3834,Z 6,A -3.2175,B 0,C 0,E1 0.1598,E2 90.0713} C_DIS
LIN {X -0.5605,Y -8.4711,Z 6,A -3.1931,B 0,C 0,E1 0.1598,E2 90.0713} C_DIS
LIN {X -0.5605,Y -8.4711,Z 6,A -3.1931,B 0,C 0,E1 0.1598,E2 90.0713} C_DIS
Enddeposition()
LIN {X 0.0002,Y -4.7528,Z 7,A -2.9998,B 0,C 0,E1 0.1598,E2 90.0603} C_DIS
Startdeposition()
$VEL.CP = VEL_PRINT
LIN {X 0.0002,Y -4.7528,Z 7,A -3.0055,B 0,C 0,E1 0.1598,E2 90.066} C_DIS
LIN {X -0.8337,Y -4.6765,Z 7,A -3.0377,B 0,C 0,E1 0.1598,E2 90.0709} C_DIS
LIN {X -1.4835,Y -4.5123,Z 7,A -3.0552,B 0,C 0,E1 0.1598,E2 90.0714} C_DIS
LIN {X -2.1048,Y -4.2605,Z 7,A -3.0674,B 0,C 0,E1 0.1598,E2 90.0714} C_DIS
LIN {X -2.6828,Y -3.9209,Z 7,A -3.0742,B 0,C 0,E1 0.1598,E2 90.0714} C_DIS
LIN {X -3.2084,Y -3.5049,Z 7,A -3.0759,B 0,C 0,E1 0.1598,E2 90.0714} C_DIS
LIN {X -3.6698,Y -3.0188,Z 7,A -3.0724,B 0,C 0,E1 0.1598,E2 90.0714} C_DIS
LIN {X -4.0579,Y -2.4722,Z 7,A -3.0635,B 0,C 0,E1 0.1598,E2 90.0714} C_DIS
LIN {X -4.3639,Y -1.8759,Z 7,A -3.0496,B 0,C 0,E1 0.1598,E2 90.0714} C_DIS
LIN {X -4.5865,Y -1.2437,Z 7,A -3.0311,B 0,C 0,E1 0.1598,E2 90.0714} C_DIS
LIN {X -4.7162,Y -0.5859,Z 7,A -3.0081,B 0,C 0,E1 0.1598,E2 90.0714} C_DIS
LIN {X -4.7491,Y 0.0836,Z 7,A -2.9811,B 0,C 0,E1 0.1598,E2 90.0714} C_DIS
LIN {X -4.6927,Y 0.7514,Z 7,A -2.9509,B 0,C 0,E1 0.1598,E2 90.0714} C_DIS
LIN {X -4.5396,Y 1.4041,Z 7,A -2.9177,B 0,C 0,E1 0.1598,E2 90.0714} C_DIS
LIN {X -4.2962,Y 2.0287,Z 7,A -2.8825,B 0,C 0,E1 0.1598,E2 90.0715} C_DIS
LIN {X -3.9669,Y 2.6127,Z 7,A -2.8458,B 0,C 0,E1 0.1598,E2 90.0716} C_DIS
LIN {X -3.5601,Y 3.1453,Z 7,A -2.8084,B 0,C 0,E1 0.1598,E2 90.0716} C_DIS
LIN {X -3.0824,Y 3.6151,Z 7,A -2.771,B 0,C 0,E1 0.1598,E2 90.0718} C_DIS
LIN {X -2.5428,Y 4.0126,Z 7,A -2.7344,B 0,C 0,E1 0.1598,E2 90.0718} C_DIS
LIN {X -1.9536,Y 4.3322,Z 7,A -2.6992,B 0,C 0,E1 0.1598,E2 90.0719} C_DIS
LIN {X -1.3238,Y 4.562,Z 7,A -2.6663,B 0,C 0,E1 0.1598,E2 90.0719} C_DIS
LIN {X -0.5022,Y 4.7227,Z 7,A -2.6293,B 0,C 0,E1 0.1598,E2 90.0721} C_DIS
LIN {X -0.0003,Y 4.752,Z 7,A -2.6095,B 0,C 0,E1 0.1598,E2 90.0721} C_DIS
LIN {X 0.6682,Y 4.704,Z 7,A -2.5869,B 0,C 0,E1 0.1598,E2 90.0721} C_DIS
LIN {X 1.3236,Y 4.5633,Z 7,A -2.5687,B 0,C 0,E1 0.1598,E2 90.0721} C_DIS
LIN {X 1.9531,Y 4.3325,Z 7,A -2.5552,B 0,C 0,E1 0.1598,E2 90.0721} C_DIS
LIN {X 2.5422,Y 4.0125,Z 7,A -2.547,B 0,C 0,E1 0.1598,E2 90.0721} C_DIS
LIN {X 3.0822,Y 3.6155,Z 7,A -2.5438,B 0,C 0,E1 0.1598,E2 90.0721} C_DIS
LIN {X 3.5597,Y 3.1455,Z 7,A -2.5461,B 0,C 0,E1 0.1598,E2 90.0721} C_DIS
LIN {X 4.0559,Y 2.4711,Z 7,A -2.5562,B 0,C 0,E1 0.1598,E2 90.0719} C_DIS
LIN {X 4.4285,Y 1.7213,Z 7,A -2.5742,B 0,C 0,E1 0.1598,E2 90.0719} C_DIS
LIN {X 4.6263,Y 1.0807,Z 7,A -2.5941,B 0,C 0,E1 0.1598,E2 90.0719} C_DIS
LIN {X 4.7311,Y 0.4188,Z 7,A -2.6183,B 0,C 0,E1 0.1598,E2 90.0719} C_DIS
LIN {X 4.7452,Y -0.2513,Z 7,A -2.6461,B 0,C 0,E1 0.1598,E2 90.0719} C_DIS
LIN {X 4.662,Y -0.9163,Z 7,A -2.6774,B 0,C 0,E1 0.1598,E2 90.0718} C_DIS
LIN {X 4.4859,Y -1.5632,Z 7,A -2.7113,B 0,C 0,E1 0.1598,E2 90.0718} C_DIS
LIN {X 4.222,Y -2.1791,Z 7,A -2.7471,B 0,C 0,E1 0.1598,E2 90.0718} C_DIS
LIN {X 3.874,Y -2.7522,Z 7,A -2.7842,B 0,C 0,E1 0.1598,E2 90.0717} C_DIS
LIN {X 3.4484,Y -3.2702,Z 7,A -2.8218,B 0,C 0,E1 0.1598,E2 90.0717} C_DIS
LIN {X 2.9529,Y -3.7217,Z 7,A -2.8592,B 0,C 0,E1 0.1598,E2 90.0717} C_DIS
LIN {X 2.4004,Y -4.1012,Z 7,A -2.8956,B 0,C 0,E1 0.1598,E2 90.0717} C_DIS
LIN {X 1.7983,Y -4.3958,Z 7,A -2.9302,B 0,C 0,E1 0.1598,E2 90.0717} C_DIS
LIN {X 1.1619,Y -4.6056,Z 7,A -2.9625,B 0,C 0,E1 0.1598,E2 90.0717} C_DIS
LIN {X 0.5024,Y -4.7253,Z 7,A -2.9918,B 0,C 0,E1 0.1598,E2 90.0716} C_DIS
LIN {X 0.5024,Y -4.7253,Z 7,A -2.9918,B 0,C 0,E1 0.1598,E2 90.0716} C_DIS
Enddeposition()
LIN {X 0.0131,Y -5.6865,Z 7,A -3.0494,B 0,C 0,E1 0.1598,E2 90.0703} C_DIS
Startdeposition()
$VEL.CP = VEL_PRINT
LIN {X 0.8713,Y -5.6226,Z 7,A -3.0163,B 0,C 0,E1 0.1598,E2 90.0715} C_DIS
LIN {X 2.3407,Y -5.187,Z 7,A -2.9438,B 0,C 0,E1 0.1598,E2 90.0715} C_DIS
LIN {X 3.5359,Y -4.4509,Z 7,A -2.8686,B 0,C 0,E1 0.1598,E2 90.0715} C_DIS
LIN {X 4.0347,Y -4.0041,Z 7,A -2.8315,B 0,C 0,E1 0.1598,E2 90.0717} C_DIS
LIN {X 4.6883,Y -3.2229,Z 7,A -2.7742,B 0,C 0,E1 0.1598,E2 90.0716} C_DIS
LIN {X 5.1204,Y -2.4691,Z 7,A -2.7264,B 0,C 0,E1 0.1598,E2 90.0716} C_DIS
LIN {X 5.3845,Y -1.8262,Z 7,A -2.6894,B 0,C 0,E1 0.1598,E2 90.0718} C_DIS
LIN {X 5.5646,Y -1.155,Z 7,A -2.6543,B 0,C 0,E1 0.1598,E2 90.0718} C_DIS
LIN {X 5.6828,Y -0.2942,Z 7,A -2.6133,B 0,C 0,E1 0.1598,E2 90.0716} C_DIS
LIN {X 5.589,Y 1.0696,Z 7,A -2.5584,B 0,C 0,E1 0.1598,E2 90.0712} C_DIS
LIN {X 5.3019,Y 2.0668,Z 7,A -2.5271,B 0,C 0,E1 0.1598,E2 90.0717} C_DIS
LIN {X 4.7911,Y 3.0598,Z 7,A -2.5038,B 0,C 0,E1 0.1598,E2 90.0717} C_DIS
LIN {X 4.3032,Y 3.7119,Z 7,A -2.4945,B 0,C 0,E1 0.1598,E2 90.072} C_DIS
LIN {X 3.7283,Y 4.2886,Z 7,A -2.4914,B 0,C 0,E1 0.1598,E2 90.072} C_DIS
LIN {X 3.0774,Y 4.7779,Z 7,A -2.4947,B 0,C 0,E1 0.1598,E2 90.0721} C_DIS
LIN {X 2.3636,Y 5.1701,Z 7,A -2.5045,B 0,C 0,E1 0.1598,E2 90.0721} C_DIS
LIN {X 1.3113,Y 5.5372,Z 7,A -2.5279,B 0,C 0,E1 0.1598,E2 90.0721} C_DIS
LIN {X 0.4839,Y 5.67,Z 7,A -2.5528,B 0,C 0,E1 0.1598,E2 90.0721} C_DIS
LIN {X -0.7842,Y 5.6366,Z 7,A -2.601,B 0,C 0,E1 0.1598,E2 90.0721} C_DIS
LIN {X -1.7191,Y 5.4178,Z 7,A -2.6447,B 0,C 0,E1 0.1598,E2 90.0721} C_DIS
LIN {X -2.4333,Y 5.1357,Z 7,A -2.6829,B 0,C 0,E1 0.1598,E2 90.072} C_DIS
LIN {X -3.1042,Y 4.7622,Z 7,A -2.7234,B 0,C 0,E1 0.1598,E2 90.0719} C_DIS
LIN {X -3.8646,Y 4.1758,Z 7,A -2.776,B 0,C 0,E1 0.1598,E2 90.0717} C_DIS
LIN {X -4.6165,Y 3.3171,Z 7,A -2.8397,B 0,C 0,E1 0.1598,E2 90.0714} C_DIS
LIN {X -5.059,Y 2.5926,Z 7,A -2.8866,B 0,C 0,E1 0.1598,E2 90.0714} C_DIS
LIN {X -5.389,Y 1.8103,Z 7,A -2.9317,B 0,C 0,E1 0.1598,E2 90.0714} C_DIS
LIN {X -5.5989,Y 0.9875,Z 7,A -2.974,B 0,C 0,E1 0.1598,E2 90.0713} C_DIS
LIN {X -5.6834,Y 0.1427,Z 7,A -3.0127,B 0,C 0,E1 0.1598,E2 90.0712} C_DIS
LIN {X -5.6415,Y -0.7054,Z 7,A -3.0468,B 0,C 0,E1 0.1598,E2 90.0712} C_DIS
LIN {X -5.4725,Y -1.5375,Z 7,A -3.0757,B 0,C 0,E1 0.1598,E2 90.0712} C_DIS
LIN {X -5.1834,Y -2.3358,Z 7,A -3.0987,B 0,C 0,E1 0.1598,E2 90.0712} C_DIS
LIN {X -4.7774,Y -3.0816,Z 7,A -3.1153,B 0,C 0,E1 0.1598,E2 90.0712} C_DIS
LIN {X -4.2646,Y -3.7583,Z 7,A -3.1251,B 0,C 0,E1 0.1598,E2 90.0712} C_DIS
LIN {X -3.6577,Y -4.3521,Z 7,A -3.1279,B 0,C 0,E1 0.1598,E2 90.0712} C_DIS
LIN {X -2.7052,Y -5.0051,Z 7,A -3.1205,B 0,C 0,E1 0.1598,E2 90.0712} C_DIS
LIN {X -1.5156,Y -5.4846,Z 7,A -3.0971,B 0,C 0,E1 0.1598,E2 90.0713} C_DIS
LIN {X -0.4588,Y -5.6658,Z 7,A -3.0661,B 0,C 0,E1 0.1598,E2 90.0715} C_DIS
LIN {X -0.4588,Y -5.6658,Z 7,A -3.0661,B 0,C 0,E1 0.1598,E2 90.0715} C_DIS
Enddeposition()
LIN {X 0.0071,Y -6.6219,Z 7,A -3.0885,B 0,C 0,E1 0.1598,E2 90.0703} C_DIS
Startdeposition()
$VEL.CP = VEL_PRINT
LIN {X -0.8572,Y -6.5643,Z 7,A -3.1189,B 0,C 0,E1 0.1598,E2 90.0714} C_DIS
LIN {X -1.5388,Y -6.4388,Z 7,A -3.1386,B 0,C 0,E1 0.1598,E2 90.0714} C_DIS
LIN {X -2.2028,Y -6.2411,Z 7,A -3.1546,B 0,C 0,E1 0.1598,E2 90.0714} C_DIS
LIN {X -2.8432,Y -5.9766,Z 7,A -3.1669,B 0,C 0,E1 0.1598,E2 90.0714} C_DIS
LIN {X -3.4529,Y -5.6473,Z 7,A -3.1754,B 0,C 0,E1 0.1598,E2 90.0713} C_DIS
LIN {X -4.0256,Y -5.2573,Z 7,A -3.1799,B 0,C 0,E1 0.1598,E2 90.0713} C_DIS
LIN {X -4.5518,Y -4.8064,Z 7,A -3.1801,B 0,C 0,E1 0.1598,E2 90.0713} C_DIS
LIN {X -5.0283,Y -4.3032,Z 7,A -3.1764,B 0,C 0,E1 0.1598,E2 90.0713} C_DIS
LIN {X -5.4506,Y -3.7539,Z 7,A -3.1687,B 0,C 0,E1 0.1598,E2 90.0712} C_DIS
LIN {X -5.8131,Y -3.1635,Z 7,A -3.1571,B 0,C 0,E1 0.1598,E2 90.0712} C_DIS
LIN {X -6.1138,Y -2.5392,Z 7,A -3.1418,B 0,C 0,E1 0.1598,E2 90.0712} C_DIS
LIN {X -6.3455,Y -1.8862,Z 7,A -3.1228,B 0,C 0,E1 0.1598,E2 90.0712} C_DIS
LIN {X -6.5081,Y -1.2127,Z 7,A -3.1004,B 0,C 0,E1 0.1598,E2 90.0712} C_DIS
LIN {X -6.6002,Y -0.5259,Z 7,A -3.0748,B 0,C 0,E1 0.1598,E2 90.0712} C_DIS
LIN {X -6.6201,Y 0.1669,Z 7,A -3.0464,B 0,C 0,E1 0.1598,E2 90.0712} C_DIS
LIN {X -6.5642,Y 0.8576,Z 7,A -3.0153,B 0,C 0,E1 0.1598,E2 90.0713} C_DIS
LIN {X -6.4386,Y 1.5391,Z 7,A -2.982,B 0,C 0,E1 0.1598,E2 90.0713} C_DIS
LIN {X -6.2432,Y 2.204,Z 7,A -2.9468,B 0,C 0,E1 0.1598,E2 90.0714} C_DIS
LIN {X -5.9794,Y 2.8448,Z 7,A -2.9101,B 0,C 0,E1 0.1598,E2 90.0714} C_DIS
LIN {X -5.6497,Y 3.4543,Z 7,A -2.8723,B 0,C 0,E1 0.1598,E2 90.0716} C_DIS
LIN {X -5.2575,Y 4.0256,Z 7,A -2.8339,B 0,C 0,E1 0.1598,E2 90.0716} C_DIS
LIN {X -4.8067,Y 4.5519,Z 7,A -2.7951,B 0,C 0,E1 0.1598,E2 90.0717} C_DIS
LIN {X -4.3047,Y 5.0298,Z 7,A -2.7565,B 0,C 0,E1 0.1598,E2 90.0717} C_DIS
LIN {X -3.7566,Y 5.4539,Z 7,A -2.7185,B 0,C 0,E1 0.1598,E2 90.0719} C_DIS
LIN {X -3.1653,Y 5.8152,Z 7,A -2.6815,B 0,C 0,E1 0.1598,E2 90.0719} C_DIS
LIN {X -2.5389,Y 6.1116,Z 7,A -2.6459,B 0,C 0,E1 0.1598,E2 90.072} C_DIS
LIN {X -1.8866,Y 6.3454,Z 7,A -2.612,B 0,C 0,E1 0.1598,E2 90.072} C_DIS
LIN {X -1.2133,Y 6.5088,Z 7,A -2.5802,B 0,C 0,E1 0.1598,E2 90.0721} C_DIS
LIN {X -0.5265,Y 6.6004,Z 7,A -2.551,B 0,C 0,E1 0.1598,E2 90.0721} C_DIS
LIN {X 0.1662,Y 6.619,Z 7,A -2.5247,B 0,C 0,E1 0.1598,E2 90.0722} C_DIS
LIN {X 0.857,Y 6.5633,Z 7,A -2.5016,B 0,C 0,E1 0.1598,E2 90.0722} C_DIS
LIN {X 1.5387,Y 6.4392,Z 7,A -2.4816,B 0,C 0,E1 0.1598,E2 90.0722} C_DIS
LIN {X 2.2034,Y 6.2434,Z 7,A -2.4654,B 0,C 0,E1 0.1598,E2 90.0722} C_DIS
LIN {X 2.8433,Y 5.9778,Z 7,A -2.4529,B 0,C 0,E1 0.1598,E2 90.0722} C_DIS
LIN {X 3.4519,Y 5.6466,Z 7,A -2.4445,B 0,C 0,E1 0.1598,E2 90.0722} C_DIS
LIN {X 4.0236,Y 5.2552,Z 7,A -2.4399,B 0,C 0,E1 0.1598,E2 90.0722} C_DIS
LIN {X 4.5525,Y 4.8074,Z 7,A -2.4393,B 0,C 0,E1 0.1598,E2 90.0722} C_DIS
LIN {X 5.0296,Y 4.3049,Z 7,A -2.443,B 0,C 0,E1 0.1598,E2 90.0722} C_DIS
LIN {X 5.4509,Y 3.7546,Z 7,A -2.4507,B 0,C 0,E1 0.1598,E2 90.0722} C_DIS
LIN {X 5.8137,Y 3.1643,Z 7,A -2.4623,B 0,C 0,E1 0.1598,E2 90.0721} C_DIS
LIN {X 6.1136,Y 2.5397,Z 7,A -2.4777,B 0,C 0,E1 0.1598,E2 90.0721} C_DIS
LIN {X 6.3453,Y 1.8867,Z 7,A -2.4968,B 0,C 0,E1 0.1598,E2 90.0721} C_DIS
LIN {X 6.5088,Y 1.2134,Z 7,A -2.5193,B 0,C 0,E1 0.1598,E2 90.072} C_DIS
LIN {X 6.5985,Y 0.5263,Z 7,A -2.5452,B 0,C 0,E1 0.1598,E2 90.072} C_DIS
LIN {X 6.6166,Y -0.1664,Z 7,A -2.5739,B 0,C 0,E1 0.1598,E2 90.0719} C_DIS
LIN {X 6.5645,Y -0.8573,Z 7,A -2.6051,B 0,C 0,E1 0.1598,E2 90.0719} C_DIS
LIN {X 6.4368,Y -1.5383,Z 7,A -2.6387,B 0,C 0,E1 0.1598,E2 90.0719} C_DIS
LIN {X 6.2415,Y -2.2031,Z 7,A -2.6741,B 0,C 0,E1 0.1598,E2 90.0718} C_DIS
LIN {X 5.9792,Y -2.8446,Z 7,A -2.711,B 0,C 0,E1 0.1598,E2 90.0718} C_DIS
LIN {X 5.6497,Y -3.4543,Z 7,A -2.749,B 0,C 0,E1 0.1598,E2 90.0718} C_DIS
LIN {X 5.2575,Y -4.0256,Z 7,A -2.7876,B 0,C 0,E1 0.1598,E2 90.0717} C_DIS
LIN {X 4.8074,Y -4.5526,Z 7,A -2.8265,B 0,C 0,E1 0.1598,E2 90.0717} C_DIS
LIN {X 4.3038,Y -5.0285,Z 7,A -2.8652,B 0,C 0,E1 0.1598,E2 90.0717} C_DIS
LIN {X 3.7561,Y -5.4531,Z 7,A -2.9034,B 0,C 0,E1 0.1598,E2 90.0717} C_DIS
LIN {X 3.165,Y -5.8147,Z 7,A -2.9404,B 0,C 0,E1 0.1598,E2 90.0716} C_DIS
LIN {X 2.5396,Y -6.1133,Z 7,A -2.976,B 0,C 0,E1 0.1598,E2 90.0716} C_DIS
LIN {X 1.8868,Y -6.3453,Z 7,A -3.0098,B 0,C 0,E1 0.1598,E2 90.0716} C_DIS
LIN {X 1.2134,Y -6.5088,Z 7,A -3.0415,B 0,C 0,E1 0.1598,E2 90.0716} C_DIS
LIN {X 0.5265,Y -6.6002,Z 7,A -3.0706,B 0,C 0,E1 0.1598,E2 90.0715} C_DIS
LIN {X 0.5265,Y -6.6002,Z 7,A -3.0706,B 0,C 0,E1 0.1598,E2 90.0715} C_DIS
Enddeposition()
LIN {X 0.0192,Y -7.554,Z 7,A -3.1286,B 0,C 0,E1 0.1598,E2 90.0703} C_DIS
Startdeposition()
$VEL.CP = VEL_PRINT
LIN {X 0.8771,Y -7.5058,Z 7,A -3.0962,B 0,C 0,E1 0.1598,E2 90.0714} C_DIS
LIN {X 1.8892,Y -7.3143,Z 7,A -3.051,B 0,C 0,E1 0.1598,E2 90.0714} C_DIS
LIN {X 3.0435,Y -6.9172,Z 7,A -2.9918,B 0,C 0,E1 0.1598,E2 90.0715} C_DIS
LIN {X 3.8215,Y -6.5212,Z 7,A -2.9464,B 0,C 0,E1 0.1598,E2 90.0715} C_DIS
LIN {X 4.6433,Y -5.9561,Z 7,A -2.8922,B 0,C 0,E1 0.1598,E2 90.0715} C_DIS
LIN {X 5.3912,Y -5.2963,Z 7,A -2.8367,B 0,C 0,E1 0.1598,E2 90.0715} C_DIS
LIN {X 5.9425,Y -4.6634,Z 7,A -2.7896,B 0,C 0,E1 0.1598,E2 90.0717} C_DIS
LIN {X 6.47,Y -3.8954,Z 7,A -2.7375,B 0,C 0,E1 0.1598,E2 90.0717} C_DIS
LIN {X 6.901,Y -3.0693,Z 7,A -2.6866,B 0,C 0,E1 0.1598,E2 90.0717} C_DIS
LIN {X 7.3145,Y -1.8977,Z 7,A -2.6213,B 0,C 0,E1 0.1598,E2 90.0714} C_DIS
LIN {X 7.4935,Y -0.9388,Z 7,A -2.5742,B 0,C 0,E1 0.1598,E2 90.0717} C_DIS
LIN {X 7.5523,Y -0.1607,Z 7,A -2.5392,B 0,C 0,E1 0.1598,E2 90.0718} C_DIS
LIN {X 7.5286,Y 0.6194,Z 7,A -2.5069,B 0,C 0,E1 0.1598,E2 90.0718} C_DIS
LIN {X 7.3887,Y 1.5849,Z 7,A -2.4708,B 0,C 0,E1 0.1598,E2 90.0717} C_DIS
LIN {X 7.028,Y 2.7818,Z 7,A -2.4331,B 0,C 0,E1 0.1598,E2 90.0715} C_DIS
LIN {X 6.314,Y 4.1549,Z 7,A -2.401,B 0,C 0,E1 0.1598,E2 90.0713} C_DIS
LIN {X 5.7019,Y 4.9589,Z 7,A -2.3901,B 0,C 0,E1 0.1598,E2 90.0719} C_DIS
LIN {X 4.7167,Y 5.9051,Z 7,A -2.3864,B 0,C 0,E1 0.1598,E2 90.0719} C_DIS
LIN {X 3.552,Y 6.6703,Z 7,A -2.3971,B 0,C 0,E1 0.1598,E2 90.072} C_DIS
LIN {X 2.2713,Y 7.2072,Z 7,A -2.4219,B 0,C 0,E1 0.1598,E2 90.0721} C_DIS
LIN {X 1.3725,Y 7.4326,Z 7,A -2.4457,B 0,C 0,E1 0.1598,E2 90.0723} C_DIS
LIN {X 0.289,Y 7.5524,Z 7,A -2.4807,B 0,C 0,E1 0.1598,E2 90.0723} C_DIS
LIN {X -0.8375,Y 7.5103,Z 7,A -2.524,B 0,C 0,E1 0.1598,E2 90.0723} C_DIS
LIN {X -1.9207,Y 7.3085,Z 7,A -2.5725,B 0,C 0,E1 0.1598,E2 90.0721} C_DIS
LIN {X -3.0852,Y 6.8947,Z 7,A -2.6329,B 0,C 0,E1 0.1598,E2 90.072} C_DIS
LIN {X -4.0341,Y 6.3899,Z 7,A -2.689,B 0,C 0,E1 0.1598,E2 90.0718} C_DIS
LIN {X -5.2006,Y 5.4753,Z 7,A -2.7704,B 0,C 0,E1 0.1598,E2 90.0715} C_DIS
LIN {X -5.7822,Y 4.8586,Z 7,A -2.8179,B 0,C 0,E1 0.1598,E2 90.0716} C_DIS
LIN {X -6.5421,Y 3.7838,Z 7,A -2.8908,B 0,C 0,E1 0.1598,E2 90.0711} C_DIS
LIN {X -7.097,Y 2.595,Z 7,A -2.9612,B 0,C 0,E1 0.1598,E2 90.071} C_DIS
LIN {X -7.3681,Y 1.6833,Z 7,A -3.0097,B 0,C 0,E1 0.1598,E2 90.0711} C_DIS
LIN {X -7.5248,Y 0.6593,Z 7,A -3.0585,B 0,C 0,E1 0.1598,E2 90.0711} C_DIS
LIN {X -7.5346,Y -0.585,Z 7,A -3.1109,B 0,C 0,E1 0.1598,E2 90.0707} C_DIS
LIN {X -7.3372,Y -1.8106,Z 7,A -3.1552,B 0,C 0,E1 0.1598,E2 90.0707} C_DIS
LIN {X -7.0353,Y -2.7475,Z 7,A -3.1839,B 0,C 0,E1 0.1598,E2 90.0709} C_DIS
LIN {X -6.5502,Y -3.7706,Z 7,A -3.2091,B 0,C 0,E1 0.1598,E2 90.0708} C_DIS
LIN {X -5.902,Y -4.7144,Z 7,A -3.2251,B 0,C 0,E1 0.1598,E2 90.0708} C_DIS
LIN {X -5.3709,Y -5.3097,Z 7,A -3.231,B 0,C 0,E1 0.1598,E2 90.0711} C_DIS
LIN {X -4.7815,Y -5.8471,Z 7,A -3.2321,B 0,C 0,E1 0.1598,E2 90.0711} C_DIS
LIN {X -4.1381,Y -6.3186,Z 7,A -3.2284,B 0,C 0,E1 0.1598,E2 90.0711} C_DIS
LIN {X -3.4489,Y -6.7204,Z 7,A -3.2201,B 0,C 0,E1 0.1598,E2 90.0711} C_DIS
LIN {X -2.4271,Y -7.1583,Z 7,A -3.2012,B 0,C 0,E1 0.1598,E2 90.0712} C_DIS
LIN {X -1.5754,Y -7.3907,Z 7,A -3.1798,B 0,C 0,E1 0.1598,E2 90.0712} C_DIS
LIN {X -0.5846,Y -7.5346,Z 7,A -3.1496,B 0,C 0,E1 0.1598,E2 90.0714} C_DIS
LIN {X -0.5846,Y -7.5346,Z 7,A -3.1496,B 0,C 0,E1 0.1598,E2 90.0714} C_DIS
Enddeposition()
LIN {X 0.0428,Y -8.4911,Z 7,A -3.1661,B 0,C 0,E1 0.1598,E2 90.0702} C_DIS
Startdeposition()
$VEL.CP = VEL_PRINT
LIN {X -0.7927,Y -8.4506,Z 7,A -3.1961,B 0,C 0,E1 0.1598,E2 90.0713} C_DIS
LIN {X -1.4563,Y -8.363,Z 7,A -3.2168,B 0,C 0,E1 0.1598,E2 90.0713} C_DIS
LIN {X -2.273,Y -8.1815,Z 7,A -3.2391,B 0,C 0,E1 0.1598,E2 90.0713} C_DIS
LIN {X -3.4004,Y -7.7775,Z 7,A -3.2632,B 0,C 0,E1 0.1598,E2 90.0711} C_DIS
LIN {X -4.1575,Y -7.4006,Z 7,A -3.2751,B 0,C 0,E1 0.1598,E2 90.0711} C_DIS
LIN {X -4.8735,Y -6.9504,Z 7,A -3.2823,B 0,C 0,E1 0.1598,E2 90.0711} C_DIS
LIN {X -5.5409,Y -6.4309,Z 7,A -3.2848,B 0,C 0,E1 0.1598,E2 90.0711} C_DIS
LIN {X -6.1528,Y -5.8471,Z 7,A -3.2826,B 0,C 0,E1 0.1598,E2 90.0711} C_DIS
LIN {X -6.7035,Y -5.2052,Z 7,A -3.2757,B 0,C 0,E1 0.1598,E2 90.071} C_DIS
LIN {X -7.188,Y -4.5121,Z 7,A -3.2643,B 0,C 0,E1 0.1598,E2 90.071} C_DIS
LIN {X -7.6004,Y -3.7738,Z 7,A -3.2483,B 0,C 0,E1 0.1598,E2 90.071} C_DIS
LIN {X -8.0158,Y -2.8016,Z 7,A -3.2223,B 0,C 0,E1 0.1598,E2 90.0707} C_DIS
LIN {X -8.3288,Y -1.6273,Z 7,A -3.1842,B 0,C 0,E1 0.1598,E2 90.0707} C_DIS
LIN {X -8.4452,Y -0.8308,Z 7,A -3.1554,B 0,C 0,E1 0.1598,E2 90.071} C_DIS
LIN {X -8.4871,Y -0.027,Z 7,A -3.1231,B 0,C 0,E1 0.1598,E2 90.071} C_DIS
LIN {X -8.451,Y 0.7771,Z 7,A -3.088,B 0,C 0,E1 0.1598,E2 90.0711} C_DIS
LIN {X -8.3034,Y 1.7722,Z 7,A -3.0404,B 0,C 0,E1 0.1598,E2 90.0709} C_DIS
LIN {X -7.9912,Y 2.8611,Z 7,A -2.9831,B 0,C 0,E1 0.1598,E2 90.0709} C_DIS
LIN {X -7.6706,Y 3.6337,Z 7,A -2.9391,B 0,C 0,E1 0.1598,E2 90.0713} C_DIS
LIN {X -7.2755,Y 4.3709,Z 7,A -2.8936,B 0,C 0,E1 0.1598,E2 90.0714} C_DIS
LIN {X -6.8099,Y 5.0657,Z 7,A -2.8473,B 0,C 0,E1 0.1598,E2 90.0715} C_DIS
LIN {X -6.2779,Y 5.7111,Z 7,A -2.8005,B 0,C 0,E1 0.1598,E2 90.0716} C_DIS
LIN {X -5.6848,Y 6.3008,Z 7,A -2.7539,B 0,C 0,E1 0.1598,E2 90.0717} C_DIS
LIN {X -5.0365,Y 6.8293,Z 7,A -2.7078,B 0,C 0,E1 0.1598,E2 90.0718} C_DIS
LIN {X -4.3398,Y 7.292,Z 7,A -2.6626,B 0,C 0,E1 0.1598,E2 90.0719} C_DIS
LIN {X -3.6007,Y 7.6836,Z 7,A -2.6189,B 0,C 0,E1 0.1598,E2 90.072} C_DIS
LIN {X -2.8269,Y 8.001,Z 7,A -2.577,B 0,C 0,E1 0.1598,E2 90.072} C_DIS
LIN {X -2.0254,Y 8.2401,Z 7,A -2.5373,B 0,C 0,E1 0.1598,E2 90.0722} C_DIS
LIN {X -1.2044,Y 8.4,Z 7,A -2.5003,B 0,C 0,E1 0.1598,E2 90.0722} C_DIS
LIN {X -0.3717,Y 8.4786,Z 7,A -2.4662,B 0,C 0,E1 0.1598,E2 90.0722} C_DIS
LIN {X 0.4647,Y 8.4752,Z 7,A -2.4355,B 0,C 0,E1 0.1598,E2 90.0723} C_DIS
LIN {X 1.2966,Y 8.3881,Z 7,A -2.4084,B 0,C 0,E1 0.1598,E2 90.0723} C_DIS
LIN {X 2.1158,Y 8.2192,Z 7,A -2.3853,B 0,C 0,E1 0.1598,E2 90.0723} C_DIS
LIN {X 2.9145,Y 7.9708,Z 7,A -2.3662,B 0,C 0,E1 0.1598,E2 90.0723} C_DIS
LIN {X 3.6847,Y 7.6444,Z 7,A -2.3515,B 0,C 0,E1 0.1598,E2 90.0723} C_DIS
LIN {X 4.4197,Y 7.2453,Z 7,A -2.3413,B 0,C 0,E1 0.1598,E2 90.0723} C_DIS
LIN {X 5.112,Y 6.7759,Z 7,A -2.3355,B 0,C 0,E1 0.1598,E2 90.0723} C_DIS
LIN {X 5.7539,Y 6.2396,Z 7,A -2.3345,B 0,C 0,E1 0.1598,E2 90.0723} C_DIS
LIN {X 6.3396,Y 5.6424,Z 7,A -2.3381,B 0,C 0,E1 0.1598,E2 90.0723} C_DIS
LIN {X 6.8639,Y 4.9906,Z 7,A -2.3464,B 0,C 0,E1 0.1598,E2 90.0722} C_DIS
LIN {X 7.3216,Y 4.2905,Z 7,A -2.3591,B 0,C 0,E1 0.1598,E2 90.0722} C_DIS
LIN {X 7.7083,Y 3.5488,Z 7,A -2.3763,B 0,C 0,E1 0.1598,E2 90.0721} C_DIS
LIN {X 8.0203,Y 2.7727,Z 7,A -2.3977,B 0,C 0,E1 0.1598,E2 90.0721} C_DIS
LIN {X 8.327,Y 1.6593,Z 7,A -2.4333,B 0,C 0,E1 0.1598,E2 90.0717} C_DIS
LIN {X 8.4655,Y 0.6301,Z 7,A -2.472,B 0,C 0,E1 0.1598,E2 90.0717} C_DIS
LIN {X 8.4857,Y -0.2003,Z 7,A -2.5066,B 0,C 0,E1 0.1598,E2 90.0718} C_DIS
LIN {X 8.4259,Y -1.0289,Z 7,A -2.544,B 0,C 0,E1 0.1598,E2 90.0718} C_DIS
LIN {X 8.2844,Y -1.8475,Z 7,A -2.584,B 0,C 0,E1 0.1598,E2 90.0718} C_DIS
LIN {X 8.0641,Y -2.6485,Z 7,A -2.6261,B 0,C 0,E1 0.1598,E2 90.0718} C_DIS
LIN {X 7.7662,Y -3.424,Z 7,A -2.6701,B 0,C 0,E1 0.1598,E2 90.0717} C_DIS
LIN {X 7.395,Y -4.1672,Z 7,A -2.7153,B 0,C 0,E1 0.1598,E2 90.0717} C_DIS
LIN {X 6.9527,Y -4.8705,Z 7,A -2.7614,B 0,C 0,E1 0.1598,E2 90.0717} C_DIS
LIN {X 6.4438,Y -5.5272,Z 7,A -2.808,B 0,C 0,E1 0.1598,E2 90.0717} C_DIS
LIN {X 5.8725,Y -6.1304,Z 7,A -2.8546,B 0,C 0,E1 0.1598,E2 90.0716} C_DIS
LIN {X 5.2447,Y -6.6745,Z 7,A -2.9008,B 0,C 0,E1 0.1598,E2 90.0716} C_DIS
LIN {X 4.5667,Y -7.1548,Z 7,A -2.9461,B 0,C 0,E1 0.1598,E2 90.0716} C_DIS
LIN {X 3.8452,Y -7.5667,Z 7,A -2.9901,B 0,C 0,E1 0.1598,E2 90.0716} C_DIS
LIN {X 3.0869,Y -7.9063,Z 7,A -3.0323,B 0,C 0,E1 0.1598,E2 90.0715} C_DIS
LIN {X 2.2992,Y -8.1702,Z 7,A -3.0724,B 0,C 0,E1 0.1598,E2 90.0715} C_DIS
LIN {X 1.4893,Y -8.3554,Z 7,A -3.1099,B 0,C 0,E1 0.1598,E2 90.0715} C_DIS
LIN {X 0.6654,Y -8.462,Z 7,A -3.1447,B 0,C 0,E1 0.1598,E2 90.0714} C_DIS
Enddeposition()
END
